(* POU FB_BACnet_RemoteAnalogValue_EX, ST *)
FUNCTION_BLOCK FB_BACnet_RemoteAnalogValue_EX
VAR_INPUT
	bEnablePV		: BOOL; (* enable present value with priority x in priority array, FALSE = priority x disable *)
	fPV		: REAL; (* decimal number for priority x, when input bEnablePV is TRUE *)
END_VAR
VAR_IN_OUT
	RemoteDevice	: FB_BACnet_RemoteDevice;
END_VAR
VAR_OUTPUT
	bReady				: BOOL;
	fPresentValue		: REAL;
	bOverridden			: BOOL;
	bOutOfService		: BOOL;
	bFault				: BOOL;
	bInAlarm			: BOOL;
	bOverRange			: BOOL;
	bUnderRange			: BOOL;
	bOtherFault			: BOOL;
	eEventState			: E_BACNETEVENTSTATE;
	bError				: BOOL;
	nErrorId			: UINT;
END_VAR
VAR CONSTANT
	nERR_NO_ERROR		: UINT := 0;
	nERR_REMOTE_DEVICE	: UINT := 1;
	nERR_WRONG_MAPPING	: UINT := 2;
	nERR_OPERATIONAL	: UINT := 3;
END_VAR
VAR
	_PresentValue AT%I*: REAL; 			(* ~(BACnet_PresentValue 				:		: )
								   			(BACnet_ObjectType 					: AV	: )
											(BACnet_RemoteCycletimeRead 		: 1000	: )
											(BACnet_RemoteFlagsRead        		: 1		: )
											(BACnet_RemoteResubscriptionInterval: 240	: )
	                                		(BACnet_RemoteCycleTimeWrite   		: 1000	: )
	                                		(BACnet_RemoteFlagsWrite       		: 1		: )	*)
    _PresentValue_Priority12 AT%Q*: REAL;(* ~(BACnet_PresentValue_Priority12		:		: )	*)
	_StatusFlags AT%I*: WORD; 			(* ~(BACnet_StatusFlags 				:		: )	*)
	_StatusFlagsBits : ST_BACnet_StatusFlags;
	_Reliability AT%I*: WORD;			(* ~(BACnet_Reliability 				:		: )	*)
	_EventState AT%I*: WORD;			(* ~(BACnet_EventState					:		: )	*)

	_nUpdateCount : UDINT := 0;
END_VAR
(* update client device *)
IF RemoteDevice._nUpdateCount = _nUpdateCount THEN
	RemoteDevice();
END_IF
(* remind current number of update counter *)
_nUpdateCount := RemoteDevice._nUpdateCount;

IF _StatusFlags < 4 THEN
	(* mapping seems to be wrong (bit string for status flags must be 4 in minimum) *)
	nErrorId := nERR_WRONG_MAPPING;

ELSIF RemoteDevice.bOperational THEN
	(* clear error flag *)
	nErrorId := nERR_NO_ERROR;
	(* ready state *)
	bReady := TRUE;

	(* write into priority array *)
	IF bEnablePV THEN
		_PresentValue_Priority12	:= fPV;
	ELSE
		_PresentValue_Priority12	:= F_BACnet_NAN();
	END_IF

	(* present value *)
	fPresentValue := _PresentValue;

	(* build bit states *)
	_StatusFlagsBits := F_BACnet_StatusFlags(_StatusFlags);

	(* copy states to output *)
	bOverridden := _StatusFlagsBits.overridden;
	bOutOfService := _StatusFlagsBits.out_of_service;
	bFault := _StatusFlagsBits.fault;
	bInAlarm := _StatusFlagsBits.in_alarm;
	bOverRange := (_Reliability = BACnetReliability_over_range);
	bUnderRange := (_Reliability = BACnetReliability_under_range);
	bOtherFault := (_Reliability = BACnetReliability_unreliable_other);
	eEventState := _EventState;
ELSIF RemoteDevice.bFirstCycle THEN
	(* first call of the server device since reboot/reset *)
	bReady := FALSE;
	_PresentValue_Priority12 := F_BACnet_NAN();
ELSE
	(* server device not ready, reset local ready also *)
	bReady := FALSE;
	(* and set error ID *)
	nErrorId := nERR_OPERATIONAL;
END_IF

(* set error flag *)
bError := (nErrorId <> nERR_NO_ERROR);
END_FUNCTION_BLOCK

(* POU FB_BACnet_RemoteAveraging, ST *)
FUNCTION_BLOCK FB_BACnet_RemoteAveraging
VAR_IN_OUT
	RemoteDevice		: FB_BACnet_RemoteDevice;
END_VAR
VAR_OUTPUT
	bReady				: BOOL;
	nAverageValue		: REAL;
	bError				: BOOL;
	nErrorId			: UINT;
END_VAR
VAR CONSTANT
	nERR_NO_ERROR		: UINT := 0;
	nERR_REMOTE_DEVICE	: UINT := 1;
	nERR_OPERATIONAL	: UINT := 3;
END_VAR
VAR
	_AverageValue AT%I*: REAL; 		(* ~(BACnet_AverageValue 				:		: )
										(BACnet_ObjectType					: AVG  	: )
										(BACnet_RemoteCycletimeRead 		: 1000	: )
										(BACnet_RemoteFlagsRead        		: 1		: )
										(BACnet_RemoteResubscriptionInterval: 240	: )
										(BACnet_RemoteCycleTimeWrite   		: 1000	: )
										(BACnet_RemoteFlagsWrite       		: 1		: )	*)

	_nUpdateCount : UDINT := 0;
END_VAR
(* update client device *)
IF RemoteDevice._nUpdateCount = _nUpdateCount THEN
	RemoteDevice();
END_IF
(* remind current number of update counter *)
_nUpdateCount := RemoteDevice._nUpdateCount;

IF RemoteDevice.bOperational THEN
	(* clear error flag *)
	nErrorId := nERR_NO_ERROR;
	(* ready state *)
	bReady := TRUE;
	(* present value *)
	nAverageValue := _AverageValue;
ELSE
	(* server device not ready, reset local ready also *)
	bReady := FALSE;
	(* and set error ID *)
	nErrorId := nERR_OPERATIONAL;
END_IF

(* set error flag *)
bError := (nErrorId <> nERR_NO_ERROR);
END_FUNCTION_BLOCK

(* POU FB_BACnet_RemoteBinaryInput, ST *)
FUNCTION_BLOCK FB_BACnet_RemoteBinaryInput
VAR_OUTPUT
	bReady				: BOOL;
	bPresentValue		: BOOL;
	bOverridden			: BOOL;
	bOutOfService		: BOOL;
	bFault				: BOOL;
	bInAlarm			: BOOL;
	bError				: BOOL;
	nErrorId			: UINT;
END_VAR
VAR CONSTANT
	nERR_NO_ERROR		: UINT := 0;
	nERR_REMOTE_DEVICE	: UINT := 1;
	nERR_WRONG_MAPPING	: UINT := 2;
	nERR_OPERATIONAL	: UINT := 3;
END_VAR
VAR_IN_OUT
	RemoteDevice			: FB_BACnet_RemoteDevice;
END_VAR
VAR
	_PresentValue AT%I*: WORD; 				(* ~(BACnet_PresentValue 				:		: )
												(BACnet_ObjectType					:BI    	: )
												(BACnet_RemoteCycletimeRead 		: 1000	: )
												(BACnet_RemoteFlagsRead        		: 1		: )
												(BACnet_RemoteResubscriptionInterval: 240	: )
		                                		(BACnet_RemoteCycleTimeWrite   		: 1000	: )
		                                		(BACnet_RemoteFlagsWrite       		: 1		: )	*)
	_StatusFlags AT%I*: WORD; 				(* ~(BACnet_StatusFlags 				:	    : )	*)
	_StatusFlagsBits : ST_BACnet_StatusFlags;

	_nUpdateCount : UDINT := 0;
END_VAR
(* update client device *)
IF RemoteDevice._nUpdateCount = _nUpdateCount THEN
	RemoteDevice();
END_IF
(* remind current number of update counter *)
_nUpdateCount := RemoteDevice._nUpdateCount;

IF _StatusFlags < 4 THEN
	(* mapping seems to be wrong (bit string for status flags must be 4 in minimum) *)
	nErrorId := nERR_WRONG_MAPPING;

ELSIF RemoteDevice.bOperational THEN
	(* clear error flag *)
	nErrorId := nERR_NO_ERROR;
	(* ready state *)
	bReady := TRUE;

	(* present value *)
	bPresentValue := F_BinPV_To_Bool(_PresentValue);

	(* build bit states *)
	_StatusFlagsBits := F_BACnet_StatusFlags(_StatusFlags);

	(* copy states to output *)
	bOverridden := _StatusFlagsBits.overridden;
	bOutOfService := _StatusFlagsBits.out_of_service;
	bFault := _StatusFlagsBits.fault;
	bInAlarm := _StatusFlagsBits.in_alarm;

ELSE
	bReady := FALSE;
	(* and set error ID *)
	nErrorId := nERR_OPERATIONAL;
END_IF

(* set error flag *)
bError := (nErrorId <> nERR_NO_ERROR);
END_FUNCTION_BLOCK

(* POU FB_BACnet_RemoteBinaryInput_EX, ST *)
FUNCTION_BLOCK FB_BACnet_RemoteBinaryInput_EX
VAR_OUTPUT
	bReady				: BOOL;
	bPresentValue		: BOOL;
	bOverridden			: BOOL;
	bOutOfService		: BOOL;
	bFault				: BOOL;
	bInAlarm			: BOOL;
	bNoSensor			: BOOL;
	bOpenLoop			: BOOL;
	bShortedLoop		: BOOL;
	bOtherFault			: BOOL;
	eEventState			: E_BACNETEVENTSTATE;
	bError				: BOOL;
	nErrorId			: UINT;
END_VAR
VAR CONSTANT
	nERR_NO_ERROR		: UINT := 0;
	nERR_REMOTE_DEVICE	: UINT := 1;
	nERR_WRONG_MAPPING	: UINT := 2;
	nERR_OPERATIONAL	: UINT := 3;
END_VAR
VAR_IN_OUT
	RemoteDevice			: FB_BACnet_RemoteDevice;
END_VAR
VAR
	_PresentValue AT%I*: WORD; 				(* ~(BACnet_PresentValue 				:		: )
												(BACnet_ObjectType					:BI    	: )
												(BACnet_RemoteCycletimeRead 		: 1000	: )
												(BACnet_RemoteFlagsRead        		: 1		: )
												(BACnet_RemoteResubscriptionInterval: 240	: )
		                                		(BACnet_RemoteCycleTimeWrite   		: 1000	: )
		                                		(BACnet_RemoteFlagsWrite       		: 1		: )	*)
	_StatusFlags AT%I*: WORD; 				(* ~(BACnet_StatusFlags 				:	    : )	*)
	_StatusFlagsBits : ST_BACnet_StatusFlags;
	_Reliability AT%I*: WORD; 				(* ~(BACnet_Reliability 				:		: )	*)
	_EventState AT%I*: WORD;				(* ~(BACnet_EventState					:		: )	*)

	_nUpdateCount : UDINT := 0;
END_VAR
(* update client device *)
IF RemoteDevice._nUpdateCount = _nUpdateCount THEN
	RemoteDevice();
END_IF
(* remind current number of update counter *)
_nUpdateCount := RemoteDevice._nUpdateCount;

IF _StatusFlags < 4 THEN
	(* mapping seems to be wrong (bit string for status flags must be 4 in minimum) *)
	nErrorId := nERR_WRONG_MAPPING;

ELSIF RemoteDevice.bOperational THEN
	(* clear error flag *)
	nErrorId := nERR_NO_ERROR;
	(* ready state *)
	bReady := TRUE;

	(* present value *)
	bPresentValue := F_BinPV_To_Bool(_PresentValue);

	(* build bit states *)
	_StatusFlagsBits := F_BACnet_StatusFlags(_StatusFlags);

	(* copy states to output *)
	bOverridden := _StatusFlagsBits.overridden;
	bOutOfService := _StatusFlagsBits.out_of_service;
	bFault := _StatusFlagsBits.fault;
	bInAlarm := _StatusFlagsBits.in_alarm;
	bNoSensor := (_Reliability = BACnetReliability_no_sensor);
	bOpenLoop := (_Reliability = BACnetReliability_open_loop);
	bShortedLoop := (_Reliability = BACnetReliability_shorted_loop);
	bOtherFault := (_Reliability = BACnetReliability_unreliable_other);
	eEventState := _EventState;

ELSE
	bReady := FALSE;
	(* and set error ID *)
	nErrorId := nERR_OPERATIONAL;
END_IF

(* set error flag *)
bError := (nErrorId <> nERR_NO_ERROR);
END_FUNCTION_BLOCK

(* POU FB_BACnet_RemoteBinaryOutput, ST *)
FUNCTION_BLOCK FB_BACnet_RemoteBinaryOutput
VAR_INPUT
	bEnablePV	: BOOL; (* enable present value with priority x in priority array, FALSE = priority x disable (NULL) *)
	bPV			: BOOL; (* present value bool type *)
END_VAR
VAR_IN_OUT
	RemoteDevice	: FB_BACnet_RemoteDevice;
END_VAR
VAR_OUTPUT
	bReady				: BOOL;
	bPresentValue		: BOOL;
	bOverridden			: BOOL;
	bOutOfService		: BOOL;
	bFault				: BOOL;
	bInAlarm			: BOOL;
	bError				: BOOL;
	nErrorId			: UINT;
END_VAR
VAR_INPUT
END_VAR
VAR CONSTANT
	nERR_NO_ERROR		: UINT := 0;
	nERR_REMOTE_DEVICE	: UINT := 1;
	nERR_WRONG_MAPPING	: UINT := 2;
	nERR_OPERATIONAL	: UINT := 3;
END_VAR
VAR
	_PresentValue AT%I*: WORD; 			(* ~(BACnet_PresentValue 				:		: )
								   			(BACnet_ObjectType 					: BO	: )
											(BACnet_RemoteCycletimeRead 		: 1000	: )
											(BACnet_RemoteFlagsRead        		: 1		: )
											(BACnet_RemoteResubscriptionInterval: 240	: )
		                            		(BACnet_RemoteCycleTimeWrite   		: 1000	: )
		                            		(BACnet_RemoteFlagsWrite       		: 1		: )	*)
    _PresentValue_Priority12 AT%Q*: WORD;(* ~(BACnet_PresentValue_Priority12		:		: )	*)
	_StatusFlags AT%I*: WORD; 			(* ~(BACnet_StatusFlags 				:		: )	*)
	_StatusFlagsBits : ST_BACnet_StatusFlags;
	_nUpdateCount : UDINT := 0;
END_VAR
(* update client device *)
IF RemoteDevice._nUpdateCount = _nUpdateCount THEN
	RemoteDevice();
END_IF
(* remind current number of update counter *)
_nUpdateCount := RemoteDevice._nUpdateCount;

IF _StatusFlags < 4 THEN
	(* mapping seems to be wrong (bit string for status flags must be 4 in minimum) *)
	nErrorId := nERR_WRONG_MAPPING;

ELSIF RemoteDevice.bOperational THEN
	(* clear error flag *)
	nErrorId := nERR_NO_ERROR;
	(* ready state *)
	bReady := TRUE;

	(* write into priority array *)
	_PresentValue_Priority12 := F_Bool_To_BinPV(bEnablePV, bPV);

	(* present value *)
	bPresentValue := F_BinPV_To_Bool(_PresentValue);

	(* build bit states *)
	_StatusFlagsBits := F_BACnet_StatusFlags(_StatusFlags);

	(* copy states to output *)
	bOverridden := _StatusFlagsBits.overridden;
	bOutOfService := _StatusFlagsBits.out_of_service;
	bFault := _StatusFlagsBits.fault;
	bInAlarm := _StatusFlagsBits.in_alarm;
ELSIF RemoteDevice.bFirstCycle THEN
	(* first call of the server device since reboot/reset *)
	bReady := FALSE;
	_PresentValue_Priority12 := BACnetBinaryPV_NULL;
ELSE
	(* server device not ready, reset local ready also *)
	bReady := FALSE;
	(* and set error ID *)
	nErrorId := nERR_OPERATIONAL;
END_IF

(* set error flag *)
bError := (nErrorId <> nERR_NO_ERROR);
END_FUNCTION_BLOCK

(* POU FB_BACnet_RemoteBinaryOutput_EX, ST *)
FUNCTION_BLOCK FB_BACnet_RemoteBinaryOutput_EX
VAR_INPUT
	bEnablePV	: BOOL; (* enable present value with priority x in priority array, FALSE = priority x disable (NULL) *)
	bPV			: BOOL; (* present value bool type *)
END_VAR
VAR_IN_OUT
	RemoteDevice	: FB_BACnet_RemoteDevice;
END_VAR
VAR_OUTPUT
	bReady				: BOOL;
	bPresentValue		: BOOL;
	bOverridden			: BOOL;
	bOutOfService		: BOOL;
	bFault				: BOOL;
	bInAlarm			: BOOL;
	bNoOutput			: BOOL;
	bOpenLoop			: BOOL;
	bShortedLoop		: BOOL;
	bOtherFault			: BOOL;
	eEventState			: E_BACNETEVENTSTATE;
	bError				: BOOL;
	nErrorId			: UINT;
END_VAR
VAR_INPUT
END_VAR
VAR CONSTANT
	nERR_NO_ERROR		: UINT := 0;
	nERR_REMOTE_DEVICE	: UINT := 1;
	nERR_WRONG_MAPPING	: UINT := 2;
	nERR_OPERATIONAL	: UINT := 3;
END_VAR
VAR
	_PresentValue AT%I*: WORD; 			(* ~(BACnet_PresentValue 				:		: )
								   			(BACnet_ObjectType 					: BO	: )
											(BACnet_RemoteCycletimeRead 		: 1000	: )
											(BACnet_RemoteFlagsRead        		: 1		: )
											(BACnet_RemoteResubscriptionInterval: 240	: )
		                            		(BACnet_RemoteCycleTimeWrite   		: 1000	: )
		                            		(BACnet_RemoteFlagsWrite       		: 1		: )	*)
    _PresentValue_Priority12 AT%Q*: WORD;(* ~(BACnet_PresentValue_Priority12		:		: )	*)
	_StatusFlags AT%I*: WORD; 			(* ~(BACnet_StatusFlags 				:		: )	*)
	_StatusFlagsBits : ST_BACnet_StatusFlags;
	_Reliability AT%I*: WORD;			(* ~(BACnet_Reliability 				:		: )	*)
	_EventState AT%I*: WORD;			(* ~(BACnet_EventState					:		: )	*)

	_nUpdateCount : UDINT := 0;
END_VAR
(* update client device *)
IF RemoteDevice._nUpdateCount = _nUpdateCount THEN
	RemoteDevice();
END_IF
(* remind current number of update counter *)
_nUpdateCount := RemoteDevice._nUpdateCount;

IF _StatusFlags < 4 THEN
	(* mapping seems to be wrong (bit string for status flags must be 4 in minimum) *)
	nErrorId := nERR_WRONG_MAPPING;

ELSIF RemoteDevice.bOperational THEN
	(* clear error flag *)
	nErrorId := nERR_NO_ERROR;
	(* ready state *)
	bReady := TRUE;

	(* write into priority array *)
	_PresentValue_Priority12 := F_Bool_To_BinPV(bEnablePV, bPV);

	(* present value *)
	bPresentValue := F_BinPV_To_Bool(_PresentValue);

	(* build bit states *)
	_StatusFlagsBits := F_BACnet_StatusFlags(_StatusFlags);

	(* copy states to output *)
	bOverridden := _StatusFlagsBits.overridden;
	bOutOfService := _StatusFlagsBits.out_of_service;
	bFault := _StatusFlagsBits.fault;
	bInAlarm := _StatusFlagsBits.in_alarm;
	bNoOutput := (_Reliability = BACnetReliability_no_output);
	bOpenLoop := (_Reliability = BACnetReliability_open_loop);
	bShortedLoop := (_Reliability = BACnetReliability_shorted_loop);
	bOtherFault := (_Reliability = BACnetReliability_unreliable_other);
	eEventState := _EventState;
ELSIF RemoteDevice.bFirstCycle THEN
	(* first call of the server device since reboot/reset *)
	bReady := FALSE;
	_PresentValue_Priority12 := BACnetBinaryPV_NULL;
ELSE
	(* server device not ready, reset local ready also *)
	bReady := FALSE;
	(* and set error ID *)
	nErrorId := nERR_OPERATIONAL;
END_IF

(* set error flag *)
bError := (nErrorId <> nERR_NO_ERROR);
END_FUNCTION_BLOCK

(* POU FB_BACnet_RemoteBinaryValue, ST *)
FUNCTION_BLOCK FB_BACnet_RemoteBinaryValue
VAR_INPUT
	bEnablePV	: BOOL; (* enable present value with priority x in priority array, FALSE = priority x disable (NULL) *)
	bPV			: BOOL; (* present value bool type *)
END_VAR
VAR_IN_OUT
	RemoteDevice		: FB_BACnet_RemoteDevice;
END_VAR
VAR_OUTPUT
	bReady				: BOOL;
	bPresentValue		: BOOL;
	bOverridden			: BOOL;
	bOutOfService		: BOOL;
	bFault				: BOOL;
	bInAlarm			: BOOL;
	bError				: BOOL;
	nErrorId			: UINT;
END_VAR
VAR CONSTANT
	nERR_NO_ERROR		: UINT := 0;
	nERR_REMOTE_DEVICE	: UINT := 1;
	nERR_WRONG_MAPPING	: UINT := 2;
	nERR_OPERATIONAL	: UINT := 3;
END_VAR
VAR

	_PresentValue AT%I*: WORD; 			(* ~(BACnet_PresentValue 				:		: )
								   			(BACnet_ObjectType 					: BV	: )
											(BACnet_RemoteCycletimeRead 		: 1000	: )
											(BACnet_RemoteFlagsRead        		: 1		: )
											(BACnet_RemoteResubscriptionInterval: 240	: )
	                                		(BACnet_RemoteCycleTimeWrite   		: 1000	: )
	                                		(BACnet_RemoteFlagsWrite       		: 1		: )	*)
    _PresentValue_Priority12 AT%Q*: WORD;(* ~(BACnet_PresentValue_Priority12		:		: )	*)
	_StatusFlags AT%I*: WORD; 			(* ~(BACnet_StatusFlags 				:		: )	*)
	_StatusFlagsBits : ST_BACnet_StatusFlags;

	_nUpdateCount : UDINT := 0;
END_VAR
(* update client device *)
IF RemoteDevice._nUpdateCount = _nUpdateCount THEN
	RemoteDevice();
END_IF
(* remind current number of update counter *)
_nUpdateCount := RemoteDevice._nUpdateCount;

IF _StatusFlags < 4 THEN
	(* mapping seems to be wrong (bit string for status flags must be 4 in minimum) *)
	nErrorId := nERR_WRONG_MAPPING;

ELSIF RemoteDevice.bOperational THEN
	(* clear error flag *)
	nErrorId := nERR_NO_ERROR;
	(* ready state *)
	bReady := TRUE;

	(* write into priority array *)
	_PresentValue_Priority12 := F_Bool_To_BinPV(bEnablePV, bPV);

	(* present value *)
	bPresentValue := F_BinPV_To_Bool(_PresentValue);

	(* build bit states *)
	_StatusFlagsBits := F_BACnet_StatusFlags(_StatusFlags);

	(* copy states to output *)
	bOverridden := _StatusFlagsBits.overridden;
	bOutOfService := _StatusFlagsBits.out_of_service;
	bFault := _StatusFlagsBits.fault;
	bInAlarm := _StatusFlagsBits.in_alarm;

ELSIF RemoteDevice.bFirstCycle THEN
	(* first call of the server device since reboot/reset *)
	bReady := FALSE;
	_PresentValue_Priority12 := BACnetBinaryPV_NULL;
ELSE
	(* server device not ready, reset local ready also *)
	bReady := FALSE;
	(* and set error ID *)
	nErrorId := nERR_OPERATIONAL;
END_IF

(* set error flag *)
bError := (nErrorId <> nERR_NO_ERROR);
END_FUNCTION_BLOCK

(* POU FB_BACnet_RemoteBinaryValue_EX, ST *)
FUNCTION_BLOCK FB_BACnet_RemoteBinaryValue_EX
VAR_INPUT
	bEnablePV	: BOOL; (* enable present value with priority x in priority array, FALSE = priority x disable (NULL) *)
	bPV			: BOOL; (* present value bool type *)
END_VAR
VAR_IN_OUT
	RemoteDevice		: FB_BACnet_RemoteDevice;
END_VAR
VAR_OUTPUT
	bReady				: BOOL;
	bPresentValue		: BOOL;
	bOverridden			: BOOL;
	bOutOfService		: BOOL;
	bFault				: BOOL;
	bInAlarm			: BOOL;
	bOtherFault			: BOOL;
	eEventState			: E_BACNETEVENTSTATE;
	bError				: BOOL;
	nErrorId			: UINT;
END_VAR
VAR CONSTANT
	nERR_NO_ERROR		: UINT := 0;
	nERR_REMOTE_DEVICE	: UINT := 1;
	nERR_WRONG_MAPPING	: UINT := 2;
	nERR_OPERATIONAL	: UINT := 3;
END_VAR
VAR

	_PresentValue AT%I*: WORD; 			(* ~(BACnet_PresentValue 				:		: )
								   			(BACnet_ObjectType 					: BV	: )
											(BACnet_RemoteCycletimeRead 		: 1000	: )
											(BACnet_RemoteFlagsRead        		: 1		: )
											(BACnet_RemoteResubscriptionInterval: 240	: )
	                                		(BACnet_RemoteCycleTimeWrite   		: 1000	: )
	                                		(BACnet_RemoteFlagsWrite       		: 1		: )	*)
    _PresentValue_Priority12 AT%Q*: WORD;(* ~(BACnet_PresentValue_Priority12		:		: )	*)
	_StatusFlags AT%I*: WORD; 			(* ~(BACnet_StatusFlags 				:		: )	*)
	_StatusFlagsBits : ST_BACnet_StatusFlags;
	_Reliability AT%I*: WORD;			(* ~(BACnet_Reliability 				:		: )	*)
	_EventState AT%I*: WORD;			(* ~(BACnet_EventState					:		: )	*)

	_nUpdateCount : UDINT := 0;
END_VAR
(* update client device *)
IF RemoteDevice._nUpdateCount = _nUpdateCount THEN
	RemoteDevice();
END_IF
(* remind current number of update counter *)
_nUpdateCount := RemoteDevice._nUpdateCount;

IF _StatusFlags < 4 THEN
	(* mapping seems to be wrong (bit string for status flags must be 4 in minimum) *)
	nErrorId := nERR_WRONG_MAPPING;

ELSIF RemoteDevice.bOperational THEN
	(* clear error flag *)
	nErrorId := nERR_NO_ERROR;
	(* ready state *)
	bReady := TRUE;

	(* write into priority array *)
	_PresentValue_Priority12 := F_Bool_To_BinPV(bEnablePV, bPV);

	(* present value *)
	bPresentValue := F_BinPV_To_Bool(_PresentValue);

	(* build bit states *)
	_StatusFlagsBits := F_BACnet_StatusFlags(_StatusFlags);

	(* copy states to output *)
	bOverridden := _StatusFlagsBits.overridden;
	bOutOfService := _StatusFlagsBits.out_of_service;
	bFault := _StatusFlagsBits.fault;
	bInAlarm := _StatusFlagsBits.in_alarm;
	bOtherFault := (_Reliability = BACnetReliability_unreliable_other);
	eEventState := _EventState;

ELSIF RemoteDevice.bFirstCycle THEN
	(* first call of the server device since reboot/reset *)
	bReady := FALSE;
	_PresentValue_Priority12 := BACnetBinaryPV_NULL;
ELSE
	(* server device not ready, reset local ready also *)
	bReady := FALSE;
	(* and set error ID *)
	nErrorId := nERR_OPERATIONAL;
END_IF

(* set error flag *)
bError := (nErrorId <> nERR_NO_ERROR);
END_FUNCTION_BLOCK

(* POU FB_BACnet_RemoteCalendar, ST *)
FUNCTION_BLOCK FB_BACnet_RemoteCalendar
VAR_IN_OUT
	RemoteDevice		: FB_BACnet_RemoteDevice;
END_VAR
VAR_OUTPUT
	bReady				: BOOL;
	bPresentValue		: BOOL;
	bError				: BOOL;
	nErrorId			: UINT;
END_VAR
VAR CONSTANT
	nERR_NO_ERROR		: UINT := 0;
	nERR_REMOTE_DEVICE	: UINT := 1;
	nERR_OPERATIONAL	: UINT := 3;
END_VAR
VAR
	_PresentValue AT%I*: BOOL;	(* ~(BACnet_PresentValue 				:		: )
									(BACnet_ObjectType 					: CAL	: )
									(BACnet_RemoteCycletimeRead 		: 1000	: )
									(BACnet_RemoteFlagsRead        		: 1		: )
									(BACnet_RemoteResubscriptionInterval: 240	: )
                            		(BACnet_RemoteCycleTimeWrite   		: 1000	: )
                            		(BACnet_RemoteFlagsWrite       		: 1		: )	*)
	_nUpdateCount : UDINT := 0;
END_VAR
(* update client device *)
IF RemoteDevice._nUpdateCount = _nUpdateCount THEN
	RemoteDevice();
END_IF
(* remind current number of update counter *)
_nUpdateCount := RemoteDevice._nUpdateCount;

IF RemoteDevice.bOperational THEN
	(* clear error flag *)
	nErrorId := nERR_NO_ERROR;
	(* ready state *)
	bReady := TRUE;
	(* present value *)
	bPresentValue := _PresentValue;
ELSE
	(* server device not ready, reset local ready also *)
	bReady := FALSE;
	(* and set error ID *)
	nErrorId := nERR_OPERATIONAL;
END_IF

(* set error flag *)
bError := (nErrorId <> nERR_NO_ERROR);
END_FUNCTION_BLOCK

(* POU FB_BACnet_RemoteCommand, ST *)
FUNCTION_BLOCK FB_BACnet_RemoteCommand
VAR_INPUT
	bEnablePV			: BOOL;
	nPV					: UDINT;
	bRetrigger			: BOOL; (* execute selected action on raising edge again *)
END_VAR
VAR_IN_OUT
	RemoteDevice		: FB_BACnet_RemoteDevice;
END_VAR
VAR_OUTPUT
	bReady				: BOOL;
	nPresentValue		: UDINT;
	bAllWritesOk		: BOOL; (* all actions in selected action list are written *)
	bInProcess			: BOOL; (* object is busy *)
	bError				: BOOL;
	nErrorId			: UINT;
END_VAR
VAR CONSTANT
	nERR_NO_ERROR		: UINT := 0;
	nERR_REMOTE_DEVICE	: UINT := 1;
	nERR_OPERATIONAL	: UINT := 3;
END_VAR
VAR
	_PresentValueIn AT%I*: UDINT; 		(* ~(BACnet_PresentValue 				:		: )
								   			(BACnet_ObjectType 					: CMD	: )
											(BACnet_RemoteCycletimeRead 		: 1000	: )
											(BACnet_RemoteFlagsRead        		: 1		: )
											(BACnet_RemoteResubscriptionInterval: 240	: )
	                                		(BACnet_RemoteCycleTimeWrite   		: 1000	: )
	                                		(BACnet_RemoteFlagsWrite       		: 1		: )	*)
	_InProcess AT%I*: BOOL;				(* ~(BACnet_InProcess 					:		: )	*)
	_AllWritesSuccessful AT%I*: BOOL;	(* ~(BACnet_AllWritesSuccessful			:		: )	*)
    _PresentValueOut AT%Q*: UDINT;		(* ~(BACnet_PresentValue	 	   		:      	: )	*)
	_nUpdateCount : UDINT := 0;
	_rtrigRetriggerPv : R_TRIG;
END_VAR
(* update client device *)
IF RemoteDevice._nUpdateCount = _nUpdateCount THEN
	RemoteDevice();
END_IF
(* remind current number of update counter *)
_nUpdateCount := RemoteDevice._nUpdateCount;

(* call trigger *)
_rtrigRetriggerPv(CLK:= bRetrigger, Q=> );

IF RemoteDevice.bOperational THEN
	(* clear error flag *)
	nErrorId := nERR_NO_ERROR;
	(* ready state *)
	bReady := TRUE;
	(* present value from BACnet *)
	nPresentValue := _PresentValueIn;
	(* present value to BACnet *)
	IF bEnablePV THEN
		IF _rtrigRetriggerPv.Q THEN
			(* trigger action list *)
			_PresentValueOut := 0;
		ELSE
			(* set present value *)
			_PresentValueOut := nPV;
		END_IF
	ELSE
		(* deactivate mapped present value --> other objects can write to property *)
		_PresentValueOut := 16#FFFFFFFF;
	END_IF
	(* other states *)
	bAllWritesOk := _AllWritesSuccessful;
	bInProcess := _InProcess;
ELSIF RemoteDevice.bFirstCycle THEN
	(* first call of the server device since reboot/reset *)
	bReady := FALSE;
	_PresentValueOut := 0;
ELSE
	(* server device not ready, reset local ready also *)
	bReady := FALSE;
	(* and set error ID *)
	nErrorId := nERR_OPERATIONAL;
END_IF

(* set error flag *)
bError := (nErrorId <> nERR_NO_ERROR);
END_FUNCTION_BLOCK

(* POU FB_BACnet_RemoteEventEnrollment, ST *)
FUNCTION_BLOCK FB_BACnet_RemoteEventEnrollment
VAR_IN_OUT
	RemoteDevice		: FB_BACnet_RemoteDevice;
END_VAR
VAR_OUTPUT
	bReady				: BOOL;
	bError				: BOOL;
	nErrorId			: UINT;
END_VAR
VAR CONSTANT
	nERR_NO_ERROR		: UINT := 0;
	nERR_REMOTE_DEVICE	: UINT := 1;
	nERR_OPERATIONAL	: UINT := 3;
END_VAR
VAR
	_ObjectType: E_BACNETOBJECTTYPE;	(* ~ (BACNET_OBJECTTYPE : EE : )	*)
	_nUpdateCount : UDINT := 0;
END_VAR
_ObjectType := BACnetObjectType_EventEnrollment;
(* update client device *)
IF RemoteDevice._nUpdateCount = _nUpdateCount THEN
	RemoteDevice();
END_IF
(* remind current number of update counter *)
_nUpdateCount := RemoteDevice._nUpdateCount;

IF RemoteDevice.bOperational THEN
	(* clear error flag *)
	nErrorId := nERR_NO_ERROR;
	(* ready state *)
	bReady := TRUE;
ELSE
	(* server device not ready, reset local ready also *)
	bReady := FALSE;
	(* and set error ID *)
	nErrorId := nERR_OPERATIONAL;
END_IF

(* set error flag *)
bError := (nErrorId <> nERR_NO_ERROR);
END_FUNCTION_BLOCK

(* POU FB_BACnet_RemoteFile, ST *)
FUNCTION_BLOCK FB_BACnet_RemoteFile
VAR_IN_OUT
	RemoteDevice		: FB_BACnet_RemoteDevice;
END_VAR
VAR_OUTPUT
	bReady				: BOOL;
	fFileSize			: UDINT;
	bError				: BOOL;
	nErrorId			: UINT;
END_VAR
VAR CONSTANT
	nERR_NO_ERROR		: UINT := 0;
	nERR_REMOTE_DEVICE	: UINT := 1;
	nERR_OPERATIONAL	: UINT := 3;
END_VAR
VAR
	_FileSize 			AT%I*: UDINT; 	(* ~(BACnet_FileSize 					:		: )
					   						(BACnet_ObjectType 					: FILE	: )
											(BACnet_RemoteCycletimeRead 		: 1000	: )
											(BACnet_RemoteFlagsRead        		: 1		: )
											(BACnet_RemoteResubscriptionInterval: 240	: )
	                                		(BACnet_RemoteCycleTimeWrite   		: 1000	: )
	                                		(BACnet_RemoteFlagsWrite       		: 1		: )	*)
	_nUpdateCount		: UDINT := 0;
END_VAR
(* update client device *)
IF RemoteDevice._nUpdateCount = _nUpdateCount THEN
	RemoteDevice();
END_IF
(* remind current number of update counter *)
_nUpdateCount := RemoteDevice._nUpdateCount;

IF RemoteDevice.bOperational THEN
	(* clear error flag *)
	nErrorId := nERR_NO_ERROR;
	(* ready state *)
	bReady := TRUE;
	fFileSize := _FileSize;
ELSE
	(* server device not ready, reset local ready also *)
	bReady := FALSE;
	(* and set error ID *)
	nErrorId := nERR_OPERATIONAL;
END_IF

(* set error flag *)
bError := (nErrorId <> nERR_NO_ERROR);
END_FUNCTION_BLOCK

(* POU FB_BACnet_RemoteGroup, ST *)
FUNCTION_BLOCK FB_BACnet_RemoteGroup
VAR_IN_OUT
	RemoteDevice		: FB_BACnet_RemoteDevice;
END_VAR
VAR_OUTPUT
	bReady				: BOOL;
	bError				: BOOL;
	nErrorId			: UINT;
END_VAR
VAR CONSTANT
	nERR_NO_ERROR		: UINT := 0;
	nERR_REMOTE_DEVICE	: UINT := 1;
	nERR_OPERATIONAL	: UINT := 3;
END_VAR
VAR
	_ObjectType: E_BACNETOBJECTTYPE;	(* ~ (BACNET_OBJECTTYPE : GROUP : )	*)
	_nUpdateCount : UDINT := 0;
END_VAR
_ObjectType := BACnetObjectType_Group;
(* update client device *)
IF RemoteDevice._nUpdateCount = _nUpdateCount THEN
	RemoteDevice();
END_IF
(* remind current number of update counter *)
_nUpdateCount := RemoteDevice._nUpdateCount;

IF RemoteDevice.bOperational THEN
	(* clear error flag *)
	nErrorId := nERR_NO_ERROR;
	(* ready state *)
	bReady := TRUE;
ELSE
	(* server device not ready, reset local ready also *)
	bReady := FALSE;
	(* and set error ID *)
	nErrorId := nERR_OPERATIONAL;
END_IF

(* set error flag *)
bError := (nErrorId <> nERR_NO_ERROR);
END_FUNCTION_BLOCK

(* POU FB_BACnet_RemoteLoop, ST *)
FUNCTION_BLOCK FB_BACnet_RemoteLoop
VAR_IN_OUT
	RemoteDevice		: FB_BACnet_RemoteDevice;
END_VAR
VAR_OUTPUT
	bReady				: BOOL;
	fControlledValue	: REAL;
	fPresentValue		: REAL;
	bOverridden			: BOOL;
	bOutOfService		: BOOL;
	bFault				: BOOL;
	bInAlarm			: BOOL;
	bError				: BOOL;
	nErrorId			: UINT;
END_VAR
VAR CONSTANT
	nERR_NO_ERROR		: UINT := 0;
	nERR_REMOTE_DEVICE	: UINT := 1;
	nERR_WRONG_MAPPING	: UINT := 2;
	nERR_OPERATIONAL	: UINT := 3;
END_VAR
VAR
	_PresentValue AT%I*: REAL; 				(* ~(BACnet_PresentValue 				: 		: )
												(BACnet_ObjectType					: LOOP	: )
			                                	(BACnet_RemoteCycletimeRead 		: 1000	: )
												(BACnet_RemoteFlagsRead        		: 1     : )
                                   				(BACnet_RemoteResubscriptionInterval: 240 	: )
		                                		(BACnet_RemoteCycleTimeWrite   		: 1000	: )
		                                		(BACnet_RemoteFlagsWrite       		: 1		: )	*)
	_StatusFlagsBits : ST_BACnet_StatusFlags;
	_ControlledVariableValue AT%I*: REAL; 	(* ~(BACnet_ControlledVariableValue 	:		: )	*)
	_StatusFlags AT%I*: WORD; 				(* ~(BACnet_StatusFlags 				:		: )	*)

	_nUpdateCount : UDINT := 0;
END_VAR
(* update client device *)
IF RemoteDevice._nUpdateCount = _nUpdateCount THEN
	RemoteDevice();
END_IF
(* remind current number of update counter *)
_nUpdateCount := RemoteDevice._nUpdateCount;

IF _StatusFlags < 4 THEN
	(* mapping seems to be wrong (bit string for status flags must be 4 in minimum) *)
	nErrorId := nERR_WRONG_MAPPING;

ELSIF RemoteDevice.bOperational THEN
	(* clear error flag *)
	nErrorId := nERR_NO_ERROR;
	(* ready state *)
	bReady := TRUE;

	(* present value *)
	fPresentValue := _PresentValue;
	fControlledValue := _ControlledVariableValue;

	(* build bit states *)
	_StatusFlagsBits := F_BACnet_StatusFlags(_StatusFlags);

	(* copy states to output *)
	bOverridden := _StatusFlagsBits.overridden;
	bOutOfService := _StatusFlagsBits.out_of_service;
	bFault := _StatusFlagsBits.fault;
	bInAlarm := _StatusFlagsBits.in_alarm;
ELSE
	(* server device not ready, reset local ready also *)
	bReady := FALSE;
	(* and set error ID *)
	nErrorId := nERR_OPERATIONAL;
END_IF

(* set error flag *)
bError := (nErrorId <> nERR_NO_ERROR);
END_FUNCTION_BLOCK

(* POU FB_BACnet_RemoteLoop_EX, ST *)
FUNCTION_BLOCK FB_BACnet_RemoteLoop_EX
VAR_IN_OUT
	RemoteDevice		: FB_BACnet_RemoteDevice;
END_VAR
VAR_OUTPUT
	bReady				: BOOL;
	fControlledValue	: REAL;
	fPresentValue		: REAL;
	bOverridden			: BOOL;
	bOutOfService		: BOOL;
	bFault				: BOOL;
	bInAlarm			: BOOL;
	bOpenLoop			: BOOL;
	bOtherFault			: BOOL;
	eEventState			: E_BACNETEVENTSTATE;
	bError				: BOOL;
	nErrorId			: UINT;
END_VAR
VAR CONSTANT
	nERR_NO_ERROR		: UINT := 0;
	nERR_REMOTE_DEVICE	: UINT := 1;
	nERR_WRONG_MAPPING	: UINT := 2;
	nERR_OPERATIONAL	: UINT := 3;
END_VAR
VAR
	_PresentValue AT%I*: REAL; 				(* ~(BACnet_PresentValue 				: LP	: )
			                                	(BACnet_RemoteCycletimeRead 		: 1000	: )
												(BACnet_RemoteFlagsRead        		: 3     : )
                                   				(BACnet_RemoteResubscriptionInterval: 240 	: )
		                                		(BACnet_RemoteCycleTimeWrite   		: 1000	: )
		                                		(BACnet_RemoteFlagsWrite       		: 1		: )	*)
	_StatusFlagsBits : ST_BACnet_StatusFlags;
	_Reliability AT%I*: WORD; 				(* ~(BACnet_Reliability 				:		: )	*)
	_ControlledVariableValue AT%I*: REAL; 	(* ~(BACnet_ControlledVariableValue 	:		: )	*)
	_StatusFlags AT%I*: WORD; 				(* ~(BACnet_StatusFlags 				:		: )	*)
	_EventState AT%I*: WORD;				(* ~(BACnet_EventState					:		: )	*)

	_nUpdateCount : UDINT := 0;
END_VAR
(* update client device *)
IF RemoteDevice._nUpdateCount = _nUpdateCount THEN
	RemoteDevice();
END_IF
(* remind current number of update counter *)
_nUpdateCount := RemoteDevice._nUpdateCount;

IF _StatusFlags < 4 THEN
	(* mapping seems to be wrong (bit string for status flags must be 4 in minimum) *)
	nErrorId := nERR_WRONG_MAPPING;

ELSIF RemoteDevice.bOperational THEN
	(* clear error flag *)
	nErrorId := nERR_NO_ERROR;
	(* ready state *)
	bReady := TRUE;

	(* present value *)
	fPresentValue := _PresentValue;
	fControlledValue := _ControlledVariableValue;

	(* build bit states *)
	_StatusFlagsBits := F_BACnet_StatusFlags(_StatusFlags);

	(* copy states to output *)
	bOverridden := _StatusFlagsBits.overridden;
	bOutOfService := _StatusFlagsBits.out_of_service;
	bFault := _StatusFlagsBits.fault;
	bInAlarm := _StatusFlagsBits.in_alarm;
	bOpenLoop := (_Reliability = BACnetReliability_open_loop);
	bOtherFault := (_Reliability = BACnetReliability_unreliable_other);
	eEventState := _EventState;
ELSE
	(* server device not ready, reset local ready also *)
	bReady := FALSE;
	(* and set error ID *)
	nErrorId := nERR_OPERATIONAL;
END_IF

(* set error flag *)
bError := (nErrorId <> nERR_NO_ERROR);
END_FUNCTION_BLOCK

(* POU FB_BACnet_RemoteMultiStateInput, ST *)
FUNCTION_BLOCK FB_BACnet_RemoteMultiStateInput
VAR_IN_OUT
	RemoteDevice		: FB_BACnet_RemoteDevice;
END_VAR
VAR_OUTPUT
	bReady				: BOOL;
	nPresentValue		: UDINT;
	bOverridden			: BOOL;
	bOutOfService		: BOOL;
	bFault				: BOOL;
	bInAlarm			: BOOL;
	bError				: BOOL;
	nErrorId			: UINT;
END_VAR
VAR CONSTANT
	nERR_NO_ERROR		: UINT := 0;
	nERR_REMOTE_DEVICE	: UINT := 1;
	nERR_WRONG_MAPPING	: UINT := 2;
	nERR_OPERATIONAL	: UINT := 3;
END_VAR
VAR
	_PresentValue AT%I*: UDINT; 	(* ~(BACnet_PresentValue 				:		: )
								   		(BACnet_ObjectType 					: MI	: )
										(BACnet_RemoteCycletimeRead 		: 1000	: )
										(BACnet_RemoteFlagsRead        		: 1		: )
										(BACnet_RemoteResubscriptionInterval: 240	: )
                                		(BACnet_RemoteCycleTimeWrite   		: 1000	: )
                                		(BACnet_RemoteFlagsWrite       		: 1		: )	*)
	_StatusFlags AT%I*: WORD; 		(* ~(BACnet_StatusFlags 				:		: )	*)
	_StatusFlagsBits : ST_BACnet_StatusFlags;

	_nUpdateCount : UDINT := 0;
END_VAR
(* update client device *)
IF RemoteDevice._nUpdateCount = _nUpdateCount THEN
	RemoteDevice();
END_IF
(* remind current number of update counter *)
_nUpdateCount := RemoteDevice._nUpdateCount;

IF _StatusFlags < 4 THEN
	(* mapping seems to be wrong (bit string for status flags must be 4 in minimum) *)
	nErrorId := nERR_WRONG_MAPPING;

ELSIF RemoteDevice.bOperational THEN
	(* clear error flag *)
	nErrorId := nERR_NO_ERROR;
	(* ready state *)
	bReady := TRUE;

	(* present value *)
	nPresentValue := _PresentValue;

	(* build bit states *)
	_StatusFlagsBits := F_BACnet_StatusFlags(_StatusFlags);

	(* copy states to output *)
	bOverridden := _StatusFlagsBits.overridden;
	bOutOfService := _StatusFlagsBits.out_of_service;
	bFault := _StatusFlagsBits.fault;
	bInAlarm := _StatusFlagsBits.in_alarm;

ELSE
	(* server device not ready, reset local ready also *)
	bReady := FALSE;
	(* and set error ID *)
	nErrorId := nERR_OPERATIONAL;
END_IF

(* set error flag *)
bError := (nErrorId <> nERR_NO_ERROR);
END_FUNCTION_BLOCK

(* POU FB_BACnet_RemoteMultiStateInput_EX, ST *)
FUNCTION_BLOCK FB_BACnet_RemoteMultiStateInput_EX
VAR_IN_OUT
	RemoteDevice		: FB_BACnet_RemoteDevice;
END_VAR
VAR_OUTPUT
	bReady				: BOOL;
	nPresentValue		: UDINT;
	bOverridden			: BOOL;
	bOutOfService		: BOOL;
	bFault				: BOOL;
	bInAlarm			: BOOL;
	bOverRange			: BOOL;
	bUnderRange			: BOOL;
	bNoSensor			: BOOL;
	bOpenLoop			: BOOL;
	bShortedLoop		: BOOL;
	bMultiStateFault	: BOOL;
	bOtherFault			: BOOL;
	eEventState			: E_BACNETEVENTSTATE;
	nNbrOfStates		: UDINT;
	bError				: BOOL;
	nErrorId			: UINT;
END_VAR
VAR CONSTANT
	nERR_NO_ERROR		: UINT := 0;
	nERR_REMOTE_DEVICE	: UINT := 1;
	nERR_WRONG_MAPPING	: UINT := 2;
	nERR_OPERATIONAL	: UINT := 3;
END_VAR
VAR
	_PresentValue AT%I*: UDINT; 	(* ~(BACnet_PresentValue 				:		: )
								   		(BACnet_ObjectType 					: MI	: )
										(BACnet_RemoteCycletimeRead 		: 1000	: )
										(BACnet_RemoteFlagsRead        		: 1		: )
										(BACnet_RemoteResubscriptionInterval: 240	: )
                                		(BACnet_RemoteCycleTimeWrite   		: 1000	: )
                                		(BACnet_RemoteFlagsWrite       		: 1		: )	*)
	_StatusFlags AT%I*: WORD; 		(* ~(BACnet_StatusFlags 				:		: )	*)
	_StatusFlagsBits : ST_BACnet_StatusFlags;
	_Reliability AT%I*: WORD; 		(* ~(BACnet_Reliability 				:		: )	*)
	_NumberOfStates AT%I*: UDINT;	(* ~(BACnet_NumberOfStates				:		: )	*)
	_EventState AT%I*: WORD; 			(* ~(BACnet_EventState 					 :		: )	*)

	_nUpdateCount : UDINT := 0;
END_VAR
(* update client device *)
IF RemoteDevice._nUpdateCount = _nUpdateCount THEN
	RemoteDevice();
END_IF
(* remind current number of update counter *)
_nUpdateCount := RemoteDevice._nUpdateCount;

IF _StatusFlags < 4 THEN
	(* mapping seems to be wrong (bit string for status flags must be 4 in minimum) *)
	nErrorId := nERR_WRONG_MAPPING;

ELSIF RemoteDevice.bOperational THEN
	(* clear error flag *)
	nErrorId := nERR_NO_ERROR;
	(* ready state *)
	bReady := TRUE;

	(* present value *)
	nPresentValue := _PresentValue;

	(* build bit states *)
	_StatusFlagsBits := F_BACnet_StatusFlags(_StatusFlags);

	(* copy states to output *)
	bOverridden := _StatusFlagsBits.overridden;
	bOutOfService := _StatusFlagsBits.out_of_service;
	bFault := _StatusFlagsBits.fault;
	bInAlarm := _StatusFlagsBits.in_alarm;
	bOverRange := (_Reliability = BACnetReliability_over_range);
	bUnderRange := (_Reliability = BACnetReliability_under_range);
	bNoSensor := (_Reliability = BACnetReliability_no_sensor);
	bOpenLoop := (_Reliability = BACnetReliability_open_loop);
	bShortedLoop := (_Reliability = BACnetReliability_shorted_loop);
	bMultiStateFault := (_Reliability = BACnetReliability_multi_state_fault);
	bOtherFault := (_Reliability = BACnetReliability_unreliable_other);
	nNbrOfStates := _NumberOfStates;
	eEventState := _EventState;

ELSE
	(* server device not ready, reset local ready also *)
	bReady := FALSE;
	(* and set error ID *)
	nErrorId := nERR_OPERATIONAL;
END_IF

(* set error flag *)
bError := (nErrorId <> nERR_NO_ERROR);
END_FUNCTION_BLOCK

(* POU FB_BACnet_RemoteMultiStateOutput, ST *)
FUNCTION_BLOCK FB_BACnet_RemoteMultiStateOutput
VAR_INPUT
	bEnablePV	: BOOL; (* enable present value with priority x in priority array, FALSE = priority x disable *)
	nPV			: UDINT; (* number for priority x, when input bEnablePV is TRUE *)
END_VAR
VAR_IN_OUT
	RemoteDevice		: FB_BACnet_RemoteDevice;
END_VAR
VAR_OUTPUT
	bReady				: BOOL;
	nPresentValue		: UDINT;
	bOverridden			: BOOL;
	bOutOfService		: BOOL;
	bFault				: BOOL;
	bInAlarm			: BOOL;
	nNbrOfStates		: UDINT;
	bError				: BOOL;
	nErrorId			: UINT;
END_VAR
VAR CONSTANT
	nERR_NO_ERROR		: UINT := 0;
	nERR_REMOTE_DEVICE	: UINT := 1;
	nERR_WRONG_MAPPING	: UINT := 2;
	nERR_OPERATIONAL	: UINT := 3;
END_VAR
VAR
	_PresentValue AT%I*: UDINT; 			(* ~(BACnet_PresentValue 				:		: )
								   				(BACnet_ObjectType					: MO	: )
												(BACnet_RemoteCycletimeRead 		: 1000	: )
												(BACnet_RemoteFlagsRead        		: 1		: )
												(BACnet_RemoteResubscriptionInterval: 240	: )
		                                		(BACnet_RemoteCycleTimeWrite   		: 1000	: )
		                                		(BACnet_RemoteFlagsWrite       		: 1		: )	*)
	_StatusFlags AT%I*: WORD; 				(* ~(BACnet_StatusFlags					:		: )	*)
	_StatusFlagsBits : ST_BACnet_StatusFlags;
    _PresentValue_Priority12 AT%Q*: UDINT;	(* ~(BACnet_PresentValue_Priority12				:		: )	*)
	_NumberOfStates AT%I*: UDINT;			(* ~(BACnet_NumberOfStates				:		: )	*)

	_nUpdateCount : UDINT := 0;
END_VAR
(* update client device *)
IF RemoteDevice._nUpdateCount = _nUpdateCount THEN
	RemoteDevice();
END_IF
(* remind current number of update counter *)
_nUpdateCount := RemoteDevice._nUpdateCount;

IF _StatusFlags < 4 THEN
	(* mapping seems to be wrong (bit string for status flags must be 4 in minimum) *)
	nErrorId := nERR_WRONG_MAPPING;

ELSIF RemoteDevice.bOperational THEN
	(* clear error flag *)
	nErrorId := nERR_NO_ERROR;
	(* ready state *)
	bReady := TRUE;

	(* write into priority array *)
	IF bEnablePV THEN
		_PresentValue_Priority12	:= nPV;
	ELSE
		_PresentValue_Priority12	:= 0;
	END_IF

	(* present value *)
	nPresentValue := _PresentValue;

	(* build bit states *)
	_StatusFlagsBits := F_BACnet_StatusFlags(_StatusFlags);

	(* copy states to output *)
	bOverridden := _StatusFlagsBits.overridden;
	bOutOfService := _StatusFlagsBits.out_of_service;
	bFault := _StatusFlagsBits.fault;
	bInAlarm := _StatusFlagsBits.in_alarm;

	(* number of states *)
	nNbrOfStates := _NumberOfStates;

ELSIF RemoteDevice.bFirstCycle THEN
	(* first call of the server device since reboot/reset *)
	bReady := FALSE;
	_PresentValue_Priority12 := 0;
ELSE
	(* server device not ready, reset local ready also *)
	bReady := FALSE;
	(* and set error ID *)
	nErrorId := nERR_OPERATIONAL;
END_IF

(* set error flag *)
bError := (nErrorId <> nERR_NO_ERROR);
END_FUNCTION_BLOCK

(* POU FB_BACnet_RemoteMultiStateOutput_EX, ST *)
FUNCTION_BLOCK FB_BACnet_RemoteMultiStateOutput_EX
VAR_INPUT
	bEnablePV			: BOOL; (* enable present value with priority x in priority array, FALSE = priority x disable *)
	nPV			: UDINT; (* number for priority x, when input bEnablePV is TRUE *)
END_VAR
VAR_IN_OUT
	RemoteDevice		: FB_BACnet_RemoteDevice;
END_VAR
VAR_OUTPUT
	bReady				: BOOL;
	nPresentValue		: UDINT;
	bOverridden			: BOOL;
	bOutOfService		: BOOL;
	bFault				: BOOL;
	bInAlarm			: BOOL;
	bNoOutput			: BOOL;
	bOpenLoop			: BOOL;
	bShortedLoop		: BOOL;
	bOtherFault			: BOOL;
	eEventState			: E_BACNETEVENTSTATE;
	nActivePrio			: UINT;
	nNbrOfStates		: UDINT;
	bError				: BOOL;
	nErrorId			: UINT;
END_VAR
VAR CONSTANT
	nERR_NO_ERROR		: UINT := 0;
	nERR_REMOTE_DEVICE	: UINT := 1;
	nERR_WRONG_MAPPING	: UINT := 2;
	nERR_OPERATIONAL	: UINT := 3;
END_VAR
VAR
	_PresentValue AT%I*: UDINT; 			(* ~(BACnet_PresentValue 				:		: )
								   				(BACnet_ObjectType					: MO	: )
												(BACnet_RemoteCycletimeRead 		: 1000	: )
												(BACnet_RemoteFlagsRead        		: 1		: )
												(BACnet_RemoteResubscriptionInterval: 240	: )
		                                		(BACnet_RemoteCycleTimeWrite   		: 1000	: )
		                                		(BACnet_RemoteFlagsWrite       		: 1		: )	*)
	_StatusFlags AT%I*: WORD; 				(* ~(BACnet_StatusFlags					:		: )	*)
	_StatusFlagsBits : ST_BACnet_StatusFlags;
	_Reliability AT%I*: WORD; 				(* ~(BACnet_Reliability					:		: )	*)
    _PresentValue_Priority12 AT%Q*: UDINT;	(* ~(BACnet_PresentValue_Priority12				:		: )	*)
	_NumberOfStates AT%I*: UDINT;			(* ~(BACnet_NumberOfStates				:		: )	*)
	_ActivePriority AT%I*: UDINT; 			(* ~(BACnet_ActivePriority 				:		: )	*)
	_EventState AT%I*: WORD;				(* ~(BACnet_EventState					:		: )	*)

	_nUpdateCount : UDINT := 0;
END_VAR
(* update client device *)
IF RemoteDevice._nUpdateCount = _nUpdateCount THEN
	RemoteDevice();
END_IF
(* remind current number of update counter *)
_nUpdateCount := RemoteDevice._nUpdateCount;

IF _StatusFlags < 4 THEN
	(* mapping seems to be wrong (bit string for status flags must be 4 in minimum) *)
	nErrorId := nERR_WRONG_MAPPING;

ELSIF RemoteDevice.bOperational THEN
	(* clear error flag *)
	nErrorId := nERR_NO_ERROR;
	(* ready state *)
	bReady := TRUE;

	(* write into priority array *)
	IF bEnablePV THEN
		_PresentValue_Priority12	:= nPV;
	ELSE
		_PresentValue_Priority12	:= 0;
	END_IF

	(* present value *)
	nPresentValue := _PresentValue;

	(* build bit states *)
	_StatusFlagsBits := F_BACnet_StatusFlags(_StatusFlags);

	(* copy states to output *)
	bOverridden := _StatusFlagsBits.overridden;
	bOutOfService := _StatusFlagsBits.out_of_service;
	bFault := _StatusFlagsBits.fault;
	bInAlarm := _StatusFlagsBits.in_alarm;
	bNoOutput := (_Reliability = BACnetReliability_no_output);
	bOpenLoop := (_Reliability = BACnetReliability_open_loop);
	bShortedLoop := (_Reliability = BACnetReliability_shorted_loop);
	bOtherFault := (_Reliability = BACnetReliability_unreliable_other);
	eEventState := _EventState;

	(* copy active priority *)
	nActivePrio := UDINT_TO_UINT(_ActivePriority);

	(* number of states *)
	nNbrOfStates := _NumberOfStates;

ELSIF RemoteDevice.bFirstCycle THEN
	(* first call of the server device since reboot/reset *)
	bReady := FALSE;
	_PresentValue_Priority12 := 0;
ELSE
	(* server device not ready, reset local ready also *)
	bReady := FALSE;
	(* and set error ID *)
	nErrorId := nERR_OPERATIONAL;
END_IF

(* set error flag *)
bError := (nErrorId <> nERR_NO_ERROR);
END_FUNCTION_BLOCK

(* POU FB_BACnet_RemoteMultiStateValue, ST *)
FUNCTION_BLOCK FB_BACnet_RemoteMultiStateValue
VAR_INPUT
	bEnablePV			: BOOL; (* enable present value with priority x in priority array, FALSE = priority x disable *)
	nPV					: UDINT; (* number for priority x, when input bEnablePV is TRUE *)
END_VAR
VAR_IN_OUT
	RemoteDevice		: FB_BACnet_RemoteDevice;
END_VAR
VAR_OUTPUT
	bReady				: BOOL;
	nPresentValue		: UDINT;
	bOverridden			: BOOL;
	bOutOfService		: BOOL;
	bFault				: BOOL;
	bInAlarm			: BOOL;
	nNbrOfStates		: UDINT;
	bError				: BOOL;
	nErrorId			: UINT;
END_VAR
VAR CONSTANT
	nERR_NO_ERROR		: UINT := 0;
	nERR_REMOTE_DEVICE	: UINT := 1;
	nERR_WRONG_MAPPING	: UINT := 2;
	nERR_OPERATIONAL	: UINT := 3;
END_VAR
VAR
	_PresentValue AT%I*: UDINT; 			(* ~(BACnet_PresentValue 				:		: )
								   				(BACnet_ObjectType 					: MV	: )
												(BACnet_RemoteCycletimeRead 		: 1000	: )
												(BACnet_RemoteFlagsRead        		: 1		: )
												(BACnet_RemoteResubscriptionInterval: 240	: )
		                                		(BACnet_RemoteCycleTimeWrite   		: 1000	: )
		                                		(BACnet_RemoteFlagsWrite       		: 1		: )	*)
	_StatusFlags AT%I*: WORD; 				(* ~(BACnet_StatusFlags 				:		: )	*)
	_StatusFlagsBits : ST_BACnet_StatusFlags;
    _PresentValue_Priority12 AT%Q*: UDINT;	(* ~(BACnet_PresentValue_Priority12				:		: )	*)
	_NumberOfStates AT%I*: UDINT;			(* ~(BACnet_NumberOfStates				:		: )	*)

	_nUpdateCount : UDINT := 0;
END_VAR
(* update client device *)
IF RemoteDevice._nUpdateCount = _nUpdateCount THEN
	RemoteDevice();
END_IF
(* remind current number of update counter *)
_nUpdateCount := RemoteDevice._nUpdateCount;

IF _StatusFlags < 4 THEN
	(* mapping seems to be wrong (bit string for status flags must be 4 in minimum) *)
	nErrorId := nERR_WRONG_MAPPING;

ELSIF RemoteDevice.bOperational THEN
	(* clear error flag *)
	nErrorId := nERR_NO_ERROR;
	(* ready state *)
	bReady := TRUE;

	(* write into priority array *)
	IF bEnablePV THEN
		_PresentValue_Priority12	:= nPV;
	ELSE
		_PresentValue_Priority12	:= 0;
	END_IF

	(* present value *)
	nPresentValue := _PresentValue;

	(* build bit states *)
	_StatusFlagsBits := F_BACnet_StatusFlags(_StatusFlags);

	(* copy states to output *)
	bOverridden := _StatusFlagsBits.overridden;
	bOutOfService := _StatusFlagsBits.out_of_service;
	bFault := _StatusFlagsBits.fault;
	bInAlarm := _StatusFlagsBits.in_alarm;

	(* number of states *)
	nNbrOfStates := _NumberOfStates;

ELSIF RemoteDevice.bFirstCycle THEN
	(* first call of the server device since reboot/reset *)
	bReady := FALSE;
	_PresentValue_Priority12 := 0;
ELSE
	(* server device not ready, reset local ready also *)
	bReady := FALSE;
	(* and set error ID *)
	nErrorId := nERR_OPERATIONAL;
END_IF

(* set error flag *)
bError := (nErrorId <> nERR_NO_ERROR);
END_FUNCTION_BLOCK

(* POU FB_BACnet_RemoteMultiStateValue_EX, ST *)
FUNCTION_BLOCK FB_BACnet_RemoteMultiStateValue_EX
VAR_INPUT
	bEnablePV		: BOOL; (* enable present value with priority x in priority array, FALSE = priority x disable *)
	nPV		: UDINT; (* number for priority x, when input bEnablePV is TRUE *)
END_VAR
VAR_IN_OUT
	RemoteDevice	: FB_BACnet_RemoteDevice;
END_VAR
VAR_OUTPUT
	bReady				: BOOL;
	nPresentValue		: UDINT;
	bOverridden			: BOOL;
	bOutOfService		: BOOL;
	bFault				: BOOL;
	bInAlarm			: BOOL;
	bMultiStateFault	: BOOL;
	bOtherFault			: BOOL;
	eEventState			: E_BACNETEVENTSTATE;
	nNbrOfStates		: UDINT;
	bError				: BOOL;
	nErrorId			: UINT;
END_VAR
VAR CONSTANT
	nERR_NO_ERROR		: UINT := 0;
	nERR_REMOTE_DEVICE	: UINT := 1;
	nERR_WRONG_MAPPING	: UINT := 2;
	nERR_OPERATIONAL	: UINT := 3;
END_VAR
VAR
	_PresentValue AT%I*: UDINT; 			(* ~(BACnet_PresentValue 				:		: )
								   				(BACnet_ObjectType 					: MV	: )
												(BACnet_RemoteCycletimeRead 		: 1000	: )
												(BACnet_RemoteFlagsRead        		: 1		: )
												(BACnet_RemoteResubscriptionInterval: 240	: )
		                                		(BACnet_RemoteCycleTimeWrite   		: 1000	: )
		                                		(BACnet_RemoteFlagsWrite       		: 1		: )	*)
	_StatusFlags AT%I*: WORD; 				(* ~(BACnet_StatusFlags 				:		: )	*)
	_StatusFlagsBits : ST_BACnet_StatusFlags;
	_Reliability AT%I*: WORD;				(* ~(BACnet_Reliability 				:		: )	*)
    _PresentValue_Priority12 AT%Q*: UDINT;	(* ~(BACnet_PresentValue_Priority12				:		: )	*)
	_NumberOfStates AT%I*: UDINT;			(* ~(BACnet_NumberOfStates				:		: )	*)
	_EventState AT%I*: WORD;			(* ~(BACnet_EventState					:		: )	*)

	_nUpdateCount : UDINT := 0;
END_VAR
(* update client device *)
IF RemoteDevice._nUpdateCount = _nUpdateCount THEN
	RemoteDevice();
END_IF
(* remind current number of update counter *)
_nUpdateCount := RemoteDevice._nUpdateCount;

IF _StatusFlags < 4 THEN
	(* mapping seems to be wrong (bit string for status flags must be 4 in minimum) *)
	nErrorId := nERR_WRONG_MAPPING;

ELSIF RemoteDevice.bOperational THEN
	(* clear error flag *)
	nErrorId := nERR_NO_ERROR;
	(* ready state *)
	bReady := TRUE;

	(* write into priority array *)
	IF bEnablePV THEN
		_PresentValue_Priority12	:= nPV;
	ELSE
		_PresentValue_Priority12	:= 0;
	END_IF

	(* present value *)
	nPresentValue := _PresentValue;

	(* build bit states *)
	_StatusFlagsBits := F_BACnet_StatusFlags(_StatusFlags);

	(* copy states to output *)
	bOverridden := _StatusFlagsBits.overridden;
	bOutOfService := _StatusFlagsBits.out_of_service;
	bFault := _StatusFlagsBits.fault;
	bInAlarm := _StatusFlagsBits.in_alarm;
	bMultiStateFault := (_Reliability = BACnetReliability_multi_state_fault);
	bOtherFault := (_Reliability = BACnetReliability_unreliable_other);
	eEventState := _EventState;

	(* number of states *)
	nNbrOfStates := _NumberOfStates;

ELSIF RemoteDevice.bFirstCycle THEN
	(* first call of the server device since reboot/reset *)
	bReady := FALSE;
	_PresentValue_Priority12 := 0;
ELSE
	(* server device not ready, reset local ready also *)
	bReady := FALSE;
	(* and set error ID *)
	nErrorId := nERR_OPERATIONAL;
END_IF

(* set error flag *)
bError := (nErrorId <> nERR_NO_ERROR);
END_FUNCTION_BLOCK

(* POU FB_BACnet_RemoteNotificationClass, ST *)
FUNCTION_BLOCK FB_BACnet_RemoteNotificationClass
VAR_IN_OUT
	RemoteDevice		: FB_BACnet_RemoteDevice;
END_VAR
VAR_OUTPUT
	bReady				: BOOL;
	bError				: BOOL;
	nErrorId			: UINT;
END_VAR
VAR CONSTANT
	nERR_NO_ERROR		: UINT := 0;
	nERR_REMOTE_DEVICE	: UINT := 1;
	nERR_OPERATIONAL	: UINT := 3;
END_VAR
VAR
	_ObjectType : E_BACNETOBJECTTYPE; (* ~(BACNET_OBJECTTYPE :NC:)  *)
	_nUpdateCount : UDINT := 0;
END_VAR
_ObjectType := BACnetObjectType_NotificationClass;
(* update client device *)
IF RemoteDevice._nUpdateCount = _nUpdateCount THEN
	RemoteDevice();
END_IF
(* remind current number of update counter *)
_nUpdateCount := RemoteDevice._nUpdateCount;

IF RemoteDevice.bOperational THEN
	(* clear error flag *)
	nErrorId := nERR_NO_ERROR;
	(* ready state *)
	bReady := TRUE;
ELSE
	(* server device not ready, reset local ready also *)
	bReady := FALSE;
	(* and set error ID *)
	nErrorId := nERR_OPERATIONAL;
END_IF

(* set error flag *)
bError := (nErrorId <> nERR_NO_ERROR);
END_FUNCTION_BLOCK

(* POU FB_BACnet_RemoteProgram, ST *)
FUNCTION_BLOCK FB_BACnet_RemoteProgram
VAR_INPUT
	bEnablePV			: BOOL;
	ePV					: E_BACNETPROGRAMREQUEST;
	bRetrigger			: BOOL; (* execute selected request on raising edge again *)
END_VAR
VAR_IN_OUT
	RemoteDevice		: FB_BACnet_RemoteDevice;
END_VAR
VAR_OUTPUT
	bReady				: BOOL;
	ePrgState			: E_BACNETPROGRAMSTATE;
	ePrgReasonHalt		: E_BACNETPROGRAMERROR;
	bOverridden			: BOOL;
	bOutOfService		: BOOL;
	bFault				: BOOL;
	bInAlarm			: BOOL;
	bError				: BOOL;
	nErrorId			: UINT;
END_VAR
VAR CONSTANT
	nERR_NO_ERROR		: UINT := 0;
	nERR_REMOTE_DEVICE	: UINT := 1;
	nERR_WRONG_MAPPING	: UINT := 2;
	nERR_OPERATIONAL	: UINT := 3;
END_VAR
VAR
	_ProgramState AT%I*: WORD;			(* ~(BACnet_ProgramState 				:		: )
								   			(BACnet_ObjectType 					: PROG	: )
			                            	(BACnet_RemoteCycletimeRead 		: 1000	: )
											(BACnet_RemoteFlagsRead        		: 1    	: )
                                   			(BACnet_RemoteResubscriptionInterval: 240 	: )
	                                		(BACnet_RemoteCycleTimeWrite   		: 1000	: )
	                                		(BACnet_RemoteFlagsWrite       		: 1		: )	*)
	_ReasonForHalt AT%I*: WORD;			(* ~(BACnet_ReasonForHalt 				: 		: )	*)
	_StatusFlags AT%I*: WORD;			(* ~(BACnet_StatusFlags 				:		: )	*)
	_StatusFlagsBits : ST_BACnet_StatusFlags;
	_ProgramChangeRequest AT%Q*: WORD;
										(* ~(BACnet_ProgramChange 				:		: )	*)
	_nUpdateCount : UDINT := 0;
	_rtrigRetriggerPv : R_TRIG;
END_VAR
(* update client device *)
IF RemoteDevice._nUpdateCount = _nUpdateCount THEN
	RemoteDevice();
END_IF
(* remind current number of update counter *)
_nUpdateCount := RemoteDevice._nUpdateCount;

(* call trigger *)
_rtrigRetriggerPv(CLK:= bRetrigger, Q=> );

IF _StatusFlags < 4 THEN
	(* mapping seems to be wrong (bit string for status flags must be 4 in minimum) *)
	nErrorId := nERR_WRONG_MAPPING;

ELSIF RemoteDevice.bOperational THEN
	(* clear error flag *)
	nErrorId := nERR_NO_ERROR;

	(* ready state *)
	bReady := TRUE;

	(* decode status flags *)
	_StatusFlagsBits := F_BACnet_StatusFlags(_StatusFlags);

	(* copy states to output *)
	bOverridden := _StatusFlagsBits.overridden;
	bOutOfService := _StatusFlagsBits.out_of_service;
	bFault := _StatusFlagsBits.fault;
	bInAlarm := _StatusFlagsBits.in_alarm;

	(* present value from BACnet *)
	ePrgState := _ProgramState;
	(* present value to BACnet *)
	IF bEnablePV THEN
		IF _rtrigRetriggerPv.Q THEN
			(* trigger request *)
			_ProgramChangeRequest := 0;
		ELSE
			(* set request value *)
			_ProgramChangeRequest := ePV;
		END_IF
	ELSE
		(* deactivate mapped request value --> other objects can write to property *)
		_ProgramChangeRequest := 16#FFFF;
	END_IF
	(* other states *)
	ePrgReasonHalt := _ReasonForHalt;
ELSIF RemoteDevice.bFirstCycle THEN
	(* first call of the server device since reboot/reset *)
	bReady := FALSE;
	_ProgramChangeRequest := 0;
ELSE
	(* server device not ready, reset local ready also *)
	bReady := FALSE;
	(* and set error ID *)
	nErrorId := nERR_OPERATIONAL;
END_IF

(* set error flag *)
bError := (nErrorId <> nERR_NO_ERROR);
END_FUNCTION_BLOCK

(* POU FB_BACnet_RemoteProgram_EX, ST *)
FUNCTION_BLOCK FB_BACnet_RemoteProgram_EX
VAR_INPUT
	bEnablePV			: BOOL;
	ePV					: E_BACNETPROGRAMREQUEST;
	bRetrigger			: BOOL; (* execute selected request on raising edge again *)
END_VAR
VAR_IN_OUT
	RemoteDevice		: FB_BACnet_RemoteDevice;
END_VAR
VAR_OUTPUT
	bReady				: BOOL;
	ePrgState			: E_BACNETPROGRAMSTATE;
	ePrgChangeReq		: E_BACNETPROGRAMREQUEST;
	ePrgReasonHalt		: E_BACNETPROGRAMERROR;
	bOverridden			: BOOL;
	bOutOfService		: BOOL;
	bFault				: BOOL;
	bInAlarm			: BOOL;
	bProcessError		: BOOL;
	bOtherFault			: BOOL;
	bError				: BOOL;
	nErrorId			: UINT;
END_VAR
VAR CONSTANT
	nERR_NO_ERROR		: UINT := 0;
	nERR_REMOTE_DEVICE	: UINT := 1;
	nERR_WRONG_MAPPING	: UINT := 2;
	nERR_OPERATIONAL	: UINT := 3;
END_VAR
VAR
	_ProgramState AT%I*: WORD;			(* ~(BACnet_ProgramState 				:		: )
								   			(BACnet_ObjectType 					: PROG	: )
			                            	(BACnet_RemoteCycletimeRead 		: 1000	: )
											(BACnet_RemoteFlagsRead        		: 3    	: )
                                   			(BACnet_RemoteResubscriptionInterval: 240 	: )
	                                		(BACnet_RemoteCycleTimeWrite   		: 1000	: )
	                                		(BACnet_RemoteFlagsWrite       		: 1		: )	*)
	_ProgramChangeState AT%I*: WORD;	(* ~(BACnet_ProgramChange 				:		: )	*)
	_ReasonForHalt AT%I*: WORD;			(* ~(BACnet_ReasonForHalt 				: 		: )	*)
	_StatusFlags AT%I*: WORD;			(* ~(BACnet_StatusFlags 				:		: )	*)
	_StatusFlagsBits : ST_BACnet_StatusFlags;
	_Reliability AT%I*: WORD;			(* ~(BACnet_Reliability 				:		: )	*)
	_ProgramChangeRequest AT%Q*: WORD;
										(* ~(BACnet_ProgramChange 				:		: )	*)
	_nUpdateCount : UDINT := 0;
	_rtrigRetriggerPv : R_TRIG;
END_VAR
(* update client device *)
IF RemoteDevice._nUpdateCount = _nUpdateCount THEN
	RemoteDevice();
END_IF
(* remind current number of update counter *)
_nUpdateCount := RemoteDevice._nUpdateCount;

(* call trigger *)
_rtrigRetriggerPv(CLK:= bRetrigger, Q=> );

IF _StatusFlags < 4 THEN
	(* mapping seems to be wrong (bit string for status flags must be 4 in minimum) *)
	nErrorId := nERR_WRONG_MAPPING;

ELSIF RemoteDevice.bOperational THEN
	(* clear error flag *)
	nErrorId := nERR_NO_ERROR;

	(* ready state *)
	bReady := TRUE;

	(* decode status flags *)
	_StatusFlagsBits := F_BACnet_StatusFlags(_StatusFlags);

	(* copy states to output *)
	bOverridden := _StatusFlagsBits.overridden;
	bOutOfService := _StatusFlagsBits.out_of_service;
	bFault := _StatusFlagsBits.fault;
	bInAlarm := _StatusFlagsBits.in_alarm;
	bProcessError := (_Reliability = BACnetReliability_process_error);
	bOtherFault := (_Reliability = BACnetReliability_unreliable_other);

	(* present value from BACnet *)
	ePrgState := _ProgramState;
	(* present value to BACnet *)
	IF bEnablePV THEN
		IF _rtrigRetriggerPv.Q THEN
			(* trigger request *)
			_ProgramChangeRequest := 0;
		ELSE
			(* set request value *)
			_ProgramChangeRequest := ePV;
		END_IF
	ELSE
		(* deactivate mapped request value --> other objects can write to property *)
		_ProgramChangeRequest := 16#FFFF;
	END_IF
	(* other states *)
	ePrgReasonHalt := _ReasonForHalt;
	ePrgChangeReq := _ProgramChangeState;

ELSIF RemoteDevice.bFirstCycle THEN
	(* first call of the server device since reboot/reset *)
	bReady := FALSE;
	_ProgramChangeRequest := 0;
ELSE
	(* server device not ready, reset local ready also *)
	bReady := FALSE;
	(* and set error ID *)
	nErrorId := nERR_OPERATIONAL;
END_IF

(* set error flag *)
bError := (nErrorId <> nERR_NO_ERROR);
END_FUNCTION_BLOCK

(* POU FB_BACnet_RemotePulseConverter, ST *)
FUNCTION_BLOCK FB_BACnet_RemotePulseConverter
VAR_IN_OUT
	RemoteDevice		: FB_BACnet_RemoteDevice;
END_VAR
VAR_OUTPUT
	bReady				: BOOL;
	bOverridden			: BOOL;
	bOutOfService		: BOOL;
	bFault				: BOOL;
	bInAlarm			: BOOL;
	bError				: BOOL;
	nErrorId			: UINT;
END_VAR
VAR CONSTANT
	nERR_NO_ERROR		: UINT := 0;
	nERR_REMOTE_DEVICE	: UINT := 1;
	nERR_WRONG_MAPPING	: UINT := 2;
	nERR_OPERATIONAL	: UINT := 3;
END_VAR
VAR
	_StatusFlags AT%I*: UINT;		(* ~(BACnet_StatusFlags 				:		: )
										(BACnet_ObjectType 					: PC	: )
										(BACnet_RemoteCycletimeRead 		: 1000	: )
										(BACnet_RemoteFlagsRead        		: 1		: )
										(BACnet_RemoteResubscriptionInterval: 240	: )
                                		(BACnet_RemoteCycleTimeWrite   		: 1000	: )
                                		(BACnet_RemoteFlagsWrite       		: 1		: )	*)
	_StatusFlagsBits : ST_BACnet_StatusFlags;
	_nUpdateCount : UDINT := 0;
END_VAR
(* update client device *)
IF RemoteDevice._nUpdateCount = _nUpdateCount THEN
	RemoteDevice();
END_IF
(* remind current number of update counter *)
_nUpdateCount := RemoteDevice._nUpdateCount;

IF _StatusFlags < 4 THEN
	(* mapping seems to be wrong (bit string for status flags must be 4 in minimum) *)
	nErrorId := nERR_WRONG_MAPPING;

ELSIF RemoteDevice.bOperational THEN
	(* clear error flag *)
	nErrorId := nERR_NO_ERROR;
	(* ready state *)
	bReady := TRUE;

	(* build bit states *)
	_StatusFlagsBits := F_BACnet_StatusFlags(_StatusFlags);

	(* copy states to output *)
	bOverridden := _StatusFlagsBits.overridden;
	bOutOfService := _StatusFlagsBits.out_of_service;
	bFault := _StatusFlagsBits.fault;
	bInAlarm := _StatusFlagsBits.in_alarm;

ELSE
	(* server device not ready, reset local ready also *)
	bReady := FALSE;
	(* and set error ID *)
	nErrorId := nERR_OPERATIONAL;
END_IF

(* set error flag *)
bError := (nErrorId <> nERR_NO_ERROR);
END_FUNCTION_BLOCK

(* POU FB_BACnet_RemoteSchedule, ST *)
FUNCTION_BLOCK FB_BACnet_RemoteSchedule
VAR_IN_OUT
	RemoteDevice			: FB_BACnet_RemoteDevice;
END_VAR
VAR_OUTPUT
	bReady				: BOOL;
	bPresentValue		: BOOL;
	bOverridden			: BOOL;
	bOutOfService		: BOOL;
	bFault				: BOOL;
	bInAlarm			: BOOL;
	bError				: BOOL;
	nErrorId			: UINT;
END_VAR
VAR CONSTANT
	nERR_NO_ERROR		: UINT := 0;
	nERR_REMOTE_DEVICE	: UINT := 1;
	nERR_WRONG_MAPPING	: UINT := 2;
	nERR_OPERATIONAL	: UINT := 3;
END_VAR
VAR
	_PresentValue AT%I*: BOOL;	(* ~(BACnet_PresentValueBool 			:		: )
									(BACnet_ObjectType 					: SCHED	: )
									(BACnet_RemoteCycletimeRead 		: 1000	: )
									(BACnet_RemoteFlagsRead        		: 1		: )
									(BACnet_RemoteResubscriptionInterval: 240	: )
                            		(BACnet_RemoteCycleTimeWrite   		: 1000	: )
                            		(BACnet_RemoteFlagsWrite       		: 1		: )	*)
	_StatusFlags AT%I*: WORD; 	(* ~(BACnet_StatusFlags 				:		: )	*)
	_StatusFlagsBits : ST_BACnet_StatusFlags;

	_nUpdateCount : UDINT := 0;
END_VAR
(* update client device *)
IF RemoteDevice._nUpdateCount = _nUpdateCount THEN
	RemoteDevice();
END_IF
(* remind current number of update counter *)
_nUpdateCount := RemoteDevice._nUpdateCount;

IF _StatusFlags < 4 THEN
	(* mapping seems to be wrong (bit string for status flags must be 4 in minimum) *)
	nErrorId := nERR_WRONG_MAPPING;

ELSIF RemoteDevice.bOperational THEN
	(* clear error flag *)
	nErrorId := nERR_NO_ERROR;
	(* ready state *)
	bReady := TRUE;

	(* present value *)
	bPresentValue := _PresentValue;

	(* build bit states *)
	_StatusFlagsBits := F_BACnet_StatusFlags(_StatusFlags);

	(* copy states to output *)
	bOverridden := _StatusFlagsBits.overridden;
	bOutOfService := _StatusFlagsBits.out_of_service;
	bFault := _StatusFlagsBits.fault;
	bInAlarm := _StatusFlagsBits.in_alarm;

ELSE
	bReady := FALSE;
	(* and set error ID *)
	nErrorId := nERR_OPERATIONAL;
END_IF

(* set error flag *)
bError := (nErrorId <> nERR_NO_ERROR);
END_FUNCTION_BLOCK

(* POU FB_BACnet_RemoteSchedule_EX, ST *)
FUNCTION_BLOCK FB_BACnet_RemoteSchedule_EX
VAR_IN_OUT
	RemoteDevice			: FB_BACnet_RemoteDevice;
END_VAR
VAR_OUTPUT
	bReady				: BOOL;
	bPresentValue		: BOOL;
	bOverridden			: BOOL;
	bOutOfService		: BOOL;
	bFault				: BOOL;
	bInAlarm			: BOOL;
	bConfigError		: BOOL;
	bOtherFault			: BOOL;
	bError				: BOOL;
	nErrorId			: UINT;
END_VAR
VAR CONSTANT
	nERR_NO_ERROR		: UINT := 0;
	nERR_REMOTE_DEVICE	: UINT := 1;
	nERR_WRONG_MAPPING	: UINT := 2;
	nERR_OPERATIONAL	: UINT := 3;
END_VAR
VAR
	_PresentValue AT%I*: BOOL;	(* ~(BACnet_PresentValueBool 			:		: )
									(BACnet_ObjectType 					: SCHED	: )
									(BACnet_RemoteCycletimeRead 		: 1000	: )
									(BACnet_RemoteFlagsRead        		: 1		: )
									(BACnet_RemoteResubscriptionInterval: 240	: )
                            		(BACnet_RemoteCycleTimeWrite   		: 1000	: )
                            		(BACnet_RemoteFlagsWrite       		: 1		: )	*)
	_Reliability AT%I*: WORD; 	(* ~(BACnet_Reliability 				:		: )	*)
	_StatusFlags AT%I*: WORD; 	(* ~(BACnet_StatusFlags 				:		: )	*)
	_StatusFlagsBits : ST_BACnet_StatusFlags;

	_nUpdateCount : UDINT := 0;
END_VAR
(* update client device *)
IF RemoteDevice._nUpdateCount = _nUpdateCount THEN
	RemoteDevice();
END_IF
(* remind current number of update counter *)
_nUpdateCount := RemoteDevice._nUpdateCount;

IF _StatusFlags < 4 THEN
	(* mapping seems to be wrong (bit string for status flags must be 4 in minimum) *)
	nErrorId := nERR_WRONG_MAPPING;

ELSIF RemoteDevice.bOperational THEN
	(* clear error flag *)
	nErrorId := nERR_NO_ERROR;
	(* ready state *)
	bReady := TRUE;

	(* present value *)
	bPresentValue := _PresentValue;

	(* build bit states *)
	_StatusFlagsBits := F_BACnet_StatusFlags(_StatusFlags);

	(* copy states to output *)
	bOverridden := _StatusFlagsBits.overridden;
	bOutOfService := _StatusFlagsBits.out_of_service;
	bFault := _StatusFlagsBits.fault;
	bInAlarm := _StatusFlagsBits.in_alarm;
	bConfigError := (_Reliability = BACnetReliability_configuration_error);
	bOtherFault := (_Reliability = BACnetReliability_unreliable_other);

ELSE
	bReady := FALSE;
	(* and set error ID *)
	nErrorId := nERR_OPERATIONAL;
END_IF

(* set error flag *)
bError := (nErrorId <> nERR_NO_ERROR);
END_FUNCTION_BLOCK

(* POU FB_BACnet_RemoteTrendLog, ST *)
FUNCTION_BLOCK FB_BACnet_RemoteTrendLog
VAR_IN_OUT
	RemoteDevice			: FB_BACnet_RemoteDevice;
END_VAR
VAR_OUTPUT
	bReady				: BOOL;
	bLogEnable			: BOOL;
	nRecordCount		: UDINT;
	nTotalCount			: UDINT;
	bError				: BOOL;
	nErrorId			: UINT;
END_VAR
VAR CONSTANT
	nERR_NO_ERROR		: UINT := 0;
	nERR_REMOTE_DEVICE	: UINT := 1;
	nERR_OPERATIONAL	: UINT := 3;
END_VAR
VAR
	_RecordCount AT%I*: UDINT;		(* ~(BACnet_RecordCount					:		: )
										(BACnet_ObjectType					: TLOG	: )
										(BACnet_RemoteCycletimeRead 		: 1000	: )
										(BACnet_RemoteFlagsRead        		: 1		: )
										(BACnet_RemoteResubscriptionInterval: 240	: )
                                		(BACnet_RemoteCycleTimeWrite   		: 1000	: )
                                		(BACnet_RemoteFlagsWrite       		: 1		: )	*)
	_TotalRecordCount AT%I*: UDINT;	(* ~(BACnet_TotalRecordCount			:		: )	*)
	_LogEnable AT%I*: BOOL;			(* ~(BACnet_LogEnable					: 		: )	*)

	_nUpdateCount : UDINT := 0;
END_VAR
(* update client device *)
IF RemoteDevice._nUpdateCount = _nUpdateCount THEN
	RemoteDevice();
END_IF
(* remind current number of update counter *)
_nUpdateCount := RemoteDevice._nUpdateCount;

IF RemoteDevice.bOperational THEN
	(* clear error flag *)
	nErrorId := nERR_NO_ERROR;
	(* ready state *)
	bReady := TRUE;

	(* other states *)
	nRecordCount := _RecordCount;
	nTotalCount := _TotalRecordCount;
	bLogEnable := _LogEnable;

ELSE
	bReady := FALSE;
	(* and set error ID *)
	nErrorId := nERR_OPERATIONAL;
END_IF

(* set error flag *)
bError := (nErrorId <> nERR_NO_ERROR);
END_FUNCTION_BLOCK

(* POU FB_BACnet_RemoteTrendLog_EX, ST *)
FUNCTION_BLOCK FB_BACnet_RemoteTrendLog_EX
VAR_OUTPUT
	bReady				: BOOL;
	bLogEnable			: BOOL;
	nRecordCount		: UDINT;
	nTotalCount			: UDINT;
	eEventState			: E_BACNETEVENTSTATE;
	bError				: BOOL;
	nErrorId			: UINT;
END_VAR
VAR_IN_OUT
	RemoteDevice			: FB_BACnet_RemoteDevice;
END_VAR
VAR CONSTANT
	nERR_NO_ERROR		: UINT := 0;
	nERR_REMOTE_DEVICE	: UINT := 1;
	nERR_WRONG_MAPPING	: UINT := 2;
	nERR_OPERATIONAL	: UINT := 3;
END_VAR
VAR
	_RecordCount AT%I*: UDINT;		(* ~(BACnet_RecordCount					:		: )
										(BACnet_ObjectType					: TLOG	: )
										(BACnet_RemoteCycletimeRead 		: 1000	: )
										(BACnet_RemoteFlagsRead        		: 1		: )
										(BACnet_RemoteResubscriptionInterval: 240	: )
                                		(BACnet_RemoteCycleTimeWrite   		: 1000	: )
                                		(BACnet_RemoteFlagsWrite       		: 1		: )	*)
	_TotalRecordCount AT%I*: UDINT;	(* ~(BACnet_TotalRecordCount			:		: )	*)
	_LogEnable AT%I*: BOOL;			(* ~(BACnet_LogEnable					: 		: )	*)
	_EventState AT%I*: WORD;		(* ~(BACnet_EventState					:		: )	*)

	_nUpdateCount : UDINT := 0;
END_VAR
(* update client device *)
IF RemoteDevice._nUpdateCount = _nUpdateCount THEN
	RemoteDevice();
END_IF
(* remind current number of update counter *)
_nUpdateCount := RemoteDevice._nUpdateCount;

IF _EventState < 0 THEN
	(* mapping seems to be wrong *)
	nErrorId := nERR_WRONG_MAPPING;

ELSIF RemoteDevice.bOperational THEN
	(* clear error flag *)
	nErrorId := nERR_NO_ERROR;
	(* ready state *)
	bReady := TRUE;

	(* convert enumeration *)
	eEventState := _EventState;

	(* other states *)
	nRecordCount := _RecordCount;
	nTotalCount := _TotalRecordCount;
	bLogEnable := _LogEnable;

ELSE
	bReady := FALSE;
	(* and set error ID *)
	nErrorId := nERR_OPERATIONAL;
END_IF

(* set error flag *)
bError := (nErrorId <> nERR_NO_ERROR);
END_FUNCTION_BLOCK

(* POU FB_BACnet_Schedule, ST *)
FUNCTION_BLOCK FB_BACnet_Schedule
VAR_IN_OUT
	Device	: FB_BACnet_Device;
END_VAR
VAR_OUTPUT
	bReady			: BOOL;
	bPresentValue	: BOOL;
	bOverridden		: BOOL;
	bOutOfService	: BOOL;
	bFault			: BOOL;
	bInAlarm		: BOOL;
	bError			: BOOL;
	nErrorId		: UINT;
END_VAR
VAR
	_PresentValue AT%I*: BOOL;	(* ~(BACnet_PresentValueBool 			 :			: )
									(BACnet_ObjectType 					 : SCHED	: )	*)
	_StatusFlags AT%I*: WORD; 	(* ~(BACnet_StatusFlags 				 :			: )	*)
	_StatusFlagsBits : ST_BACnet_StatusFlags;
	_nUpdateCount : UDINT := 0;
END_VAR
VAR CONSTANT
	nERR_NO_ERROR		: UINT := 0;
	nERR_WRONG_MAPPING	: UINT := 2;
	nERR_OPERATIONAL	: UINT := 3;
END_VAR
(* update server device *)
IF Device._nUpdateCount = _nUpdateCount THEN
	Device();
END_IF
(* remind current number of update counter *)
_nUpdateCount := Device._nUpdateCount;

(* check BitString format of StatusFlags --> if StatusFlags are less than 4, object isn't linked correctly *)
IF (_StatusFlags < 4) THEN
	(* wrong mapping *)
	nErrorId := nERR_WRONG_MAPPING;
	bReady := FALSE;

ELSIF Device.bOperational THEN
	(* ready state *)
	bReady := TRUE;
	nErrorId := nERR_NO_ERROR;

	(* present value *)
	bPresentValue := _PresentValue;

	(* build bit states *)
	_StatusFlagsBits := F_BACnet_StatusFlags(_StatusFlags);

	(* copy states to output *)
	bOverridden := _StatusFlagsBits.overridden;
	bOutOfService := _StatusFlagsBits.out_of_service;
	bFault := _StatusFlagsBits.fault;
	bInAlarm := _StatusFlagsBits.in_alarm;

ELSE
	bReady := FALSE;
	nErrorId := nERR_OPERATIONAL;
END_IF
(* set error flag *)
bError := (nErrorId <> nERR_NO_ERROR);
END_FUNCTION_BLOCK

(* POU FB_BACnet_Schedule_EX, ST *)
FUNCTION_BLOCK FB_BACnet_Schedule_EX
VAR_IN_OUT
	Device	: FB_BACnet_Device;
END_VAR
VAR_OUTPUT
	bReady			: BOOL;
	bPresentValue	: BOOL;
	bOverridden		: BOOL;
	bOutOfService	: BOOL;
	bFault			: BOOL;
	bInAlarm		: BOOL;
	bConfigError	: BOOL;
	bOtherFault		: BOOL;
	bError			: BOOL;
	nErrorId		: UINT;
END_VAR
VAR
	_PresentValue AT%I*: BOOL;	(* ~(BACnet_PresentValueBool 			 :			: )
									(BACnet_ObjectType 					 : SCHED	: )	*)
	_Reliability AT%I*: WORD; 	(* ~(BACnet_Reliability 				 :			: )	*)
	_StatusFlags AT%I*: WORD; 	(* ~(BACnet_StatusFlags 				 :			: )	*)
	_StatusFlagsBits : ST_BACnet_StatusFlags;
	_nUpdateCount : UDINT := 0;
END_VAR
VAR CONSTANT
	nERR_NO_ERROR		: UINT := 0;
	nERR_WRONG_MAPPING	: UINT := 2;
	nERR_OPERATIONAL	: UINT := 3;
END_VAR
(* update server device *)
IF Device._nUpdateCount = _nUpdateCount THEN
	Device();
END_IF
(* remind current number of update counter *)
_nUpdateCount := Device._nUpdateCount;

(* check BitString format of StatusFlags --> if StatusFlags are less than 4, object isn't linked correctly *)
IF (_StatusFlags < 4) THEN
	(* wrong mapping *)
	nErrorId := nERR_WRONG_MAPPING;
	bReady := FALSE;

ELSIF Device.bOperational THEN
	(* ready state *)
	bReady := TRUE;
	nErrorId := nERR_NO_ERROR;

	(* present value *)
	bPresentValue := _PresentValue;

	(* build bit states *)
	_StatusFlagsBits := F_BACnet_StatusFlags(_StatusFlags);

	(* copy states to output *)
	bOverridden := _StatusFlagsBits.overridden;
	bOutOfService := _StatusFlagsBits.out_of_service;
	bFault := _StatusFlagsBits.fault;
	bInAlarm := _StatusFlagsBits.in_alarm;
	bConfigError := (_Reliability = BACnetReliability_configuration_error);
	bOtherFault := (_Reliability = BACnetReliability_unreliable_other);

ELSE
	bReady := FALSE;
	nErrorId := nERR_OPERATIONAL;
END_IF
(* set error flag *)
bError := (nErrorId <> nERR_NO_ERROR);
END_FUNCTION_BLOCK

(* POU FB_BACnet_TrendLog, ST *)
FUNCTION_BLOCK FB_BACnet_TrendLog
VAR_IN_OUT
	Device	: FB_BACnet_Device;
END_VAR
VAR_OUTPUT
	bReady			: BOOL;
	bLogEnable		: BOOL;
	nRecordCount	: UDINT;
	nTotalCount		: UDINT;
	bError			: BOOL;
	nErrorId		: UINT;
END_VAR
VAR
	_RecordCount AT%I*: UDINT;		(* ~(BACnet_RecordCount			:		: )
										(BACnet_ObjectType			: TLOG	: )	*)
	_TotalRecordCount AT%I*: UDINT;	(* ~(BACnet_TotalRecordCount	:		: )	*)
	_LogEnable AT%I*: BOOL;			(* ~(BACnet_LogEnable			: 		: )	*)
	_nUpdateCount : UDINT := 0;
END_VAR
VAR CONSTANT
	nERR_NO_ERROR		: UINT := 0;
	nERR_OPERATIONAL	: UINT := 3;
END_VAR
(* update server device *)
IF Device._nUpdateCount = _nUpdateCount THEN
	Device();
END_IF
(* remind current number of update counter *)
_nUpdateCount := Device._nUpdateCount;

IF Device.bOperational THEN
	(* ready state *)
	bReady := TRUE;
	nErrorId := nERR_NO_ERROR;
	bLogEnable := _LogEnable;

	(* other states *)
	nRecordCount := _RecordCount;
	nTotalCount := _TotalRecordCount;

ELSE
	bReady := FALSE;
	nErrorId := nERR_OPERATIONAL;
END_IF
(* set error flag *)
bError := (nErrorId <> nERR_NO_ERROR);
END_FUNCTION_BLOCK

(* POU FB_BACnet_TrendLog_EX, ST *)
FUNCTION_BLOCK FB_BACnet_TrendLog_EX
VAR_IN_OUT
	Device	: FB_BACnet_Device;
END_VAR
VAR_OUTPUT
	bReady			: BOOL;
	bLogEnable		: BOOL;
	nRecordCount	: UDINT;
	nTotalCount		: UDINT;
	eEventState		: E_BACNETEVENTSTATE;
	bAckedTrans_ToOffNormal : BOOL;
	bAckedTrans_ToFault		: BOOL;
	bAckedTrans_ToNormal	: BOOL;
	bError			: BOOL;
	nErrorId		: UINT;
END_VAR
VAR
	_RecordCount AT%I*: UDINT;		(* ~(BACnet_RecordCount			:		: )
										(BACnet_ObjectType			: TLOG	: )	*)
	_TotalRecordCount AT%I*: UDINT;	(* ~(BACnet_TotalRecordCount	:		: )	*)
	_LogEnable AT%I*: BOOL;			(* ~(BACnet_LogEnable			: 		: )	*)
	_EventState AT%I*: WORD;		(* ~(BACnet_EventState			:		: )	*)
	_AckedTransitions AT%I*:WORD;	(* ~(BACnet_AckedTransitions:		: ) *)
	_AckedTransBits : ST_BACnet_EventTransitionBits;
	_nUpdateCount : UDINT := 0;
END_VAR
VAR CONSTANT
	nERR_NO_ERROR		: UINT := 0;
	nERR_WRONG_MAPPING	: UINT := 2;
	nERR_OPERATIONAL	: UINT := 3;
END_VAR
(* update server device *)
IF Device._nUpdateCount = _nUpdateCount THEN
	Device();
END_IF
(* remind current number of update counter *)
_nUpdateCount := Device._nUpdateCount;

IF (_EventState < 0) OR _AckedTransitions < 5 THEN
	(* wrong mapping *)
	nErrorId := nERR_WRONG_MAPPING;
	bReady := FALSE;

ELSIF Device.bOperational THEN
	(* ready state *)
	bReady := TRUE;
	bLogEnable := _LogEnable;
	nErrorId := nERR_NO_ERROR;

	(* build bit states *)
	_AckedTransBits		:= F_BACnet_EventTransitionFlags(_AckedTransitions);
	bAckedTrans_ToOffNormal := _AckedTransBits.to_offnormal;
	bAckedTrans_ToFault := _AckedTransBits.to_fault;
	bAckedTrans_ToNormal := _AckedTransBits.to_normal;

	(* convert enumeration *)
	eEventState := _EventState;

	(* other states *)
	nRecordCount := _RecordCount;
	nTotalCount := _TotalRecordCount;

ELSE
	bReady := FALSE;
	nErrorId := nERR_OPERATIONAL;
END_IF
(* set error flag *)
bError := (nErrorId <> nERR_NO_ERROR);
END_FUNCTION_BLOCK
